// TwinCAT 3 PLC project OSCAT
// Title: AixOCAT
// Company: RWTH Aachen University; E.ON Energy Research Center
// ProjectVersion: 1.0.0
// ProgramVersion: 3.1.4022.1
// project tree:
//   beckhoff_network/Data types/DATA_LOG/ DLOG_DATA.TcDUT, LOG_CONTROL.TcDUT, MYSQL_COM.TcDUT (not stored), PRINTF_DATA.TcDUT (not stored), UNI_CIRCULAR_BUFFER_DATA.TcDUT (not stored), us_LOG_VIEWPORT.TcDUT
//   beckhoff_network/Data types/FILE_SERVER/ FILE_PATH_DATA.TcDUT, FILE_SERVER_DATA.TcDUT
//   beckhoff_network/Data types/NETWORK/ IP2GEO_DATA.TcDUT (not stored), IP_C.TcDUT (not stored), IP_FIFO_DATA.TcDUT (not stored), NETWORK_BUFFER.TcDUT, NETWORK_BUFFER_SHORT.TcDUT (not stored), NW_BUF_LONG.TcDUT (not stored), NW_BUF_SHORT.TcDUT, URL.TcDUT (not stored), VMAP_DATA.TcDUT (not stored), XML_CONTROL.TcDUT (not stored)
//   beckhoff_network/Data types/NET_VAR/ NET_VAR_DATA.TcDUT
//   beckhoff_network/Data types/TELNET_VISION/ us_TN_INPUT_CONTROL.TcDUT, us_TN_INPUT_CONTROL_DATA.TcDUT (not stored), us_TN_MENU.TcDUT, us_TN_MENU_POPUP.TcDUT (not stored), us_TN_SCREEN.TcDUT
//   beckhoff_network/Data types/WEATHER/ WORLD_WEATHER_CUR.TcDUT (not stored), WORLD_WEATHER_DATA.TcDUT, WORLD_WEATHER_DAY.TcDUT (not stored), YAHOO_WEATHER_DATA.TcDUT (not stored)
//   beckhoff_network/Global Variables/ Constants_1.TcGVL, Globale_Variablen_1.TcGVL
//   beckhoff_network/POUs/CO_NVERT/ BASE64_DECODE_STR.TcPOU, BASE64_DECODE_STREAM.TcPOU, BASE64_ENCODE_STR.TcPOU (not stored), BASE64_ENCODE_STREAM.TcPOU, HTML_DECODE.TcPOU (not stored), HTML_ENCODE.TcPOU (not stored), IP4_CHECK.TcPOU, IP4_DECODE.TcPOU (not stored), IP4_TO_STRING.TcPOU, IS_IP4.TcPOU, IS_URLCHR.TcPOU (not stored), MD5_AUX.TcPOU, MD5_CRAM_AUTH.TcPOU (not stored), MD5_STR.TcPOU (not stored), MD5_STREAM.TcPOU (not stored), MD5_TO_STRH.TcPOU, RC4_CRYPT_STREAM.TcPOU (not stored), SHA1_STR.TcPOU, SHA1_STREAM.TcPOU, SHA1_TO_STRH.TcPOU (not stored), STRING_TO_URL.TcPOU (not stored), URL_DECODE.TcPOU (not stored), URL_ENCODE.TcPOU, URL_TO_STRING.TcPOU (not stored)
//   beckhoff_network/POUs/DATA_LOG/ DLOG_BOOL.TcPOU (not stored), DLOG_DINT.TcPOU (not stored), DLOG_DT.TcPOU (not stored), DLOG_FILE_TO_FTP.TcPOU (not stored), DLOG_FILE_TO_SMTP.TcPOU (not stored), DLOG_REAL.TcPOU (not stored), DLOG_STORE_FILE_CSV.TcPOU (not stored), DLOG_STORE_FILE_HTML.TcPOU (not stored), DLOG_STORE_FILE_XML.TcPOU (not stored), DLOG_STORE_RRD.TcPOU (not stored), DLOG_STRING.TcPOU (not stored), UNI_CIRCULAR_BUFFER.TcPOU (not stored)
//   beckhoff_network/POUs/DEMO/ BASE64_DEMO.TcPOU (not stored) (excluded from build), CSV_PARSER_BUF_DEMO.TcPOU (not stored) (excluded from build), CSV_PARSER_FILE_DEMO.TcPOU (excluded from build), DLOG_FILE_CSV_DEMO.TcPOU (not stored) (excluded from build), DLOG_FILE_CSV_FTP_DEMO.TcPOU (not stored) (excluded from build), DLOG_FILE_CSV_SMTP_DEMO.TcPOU (not stored) (excluded from build), DLOG_FILE_HTML_DEMO.TcPOU (not stored) (excluded from build), DLOG_FILE_XML_DEMO.TcPOU (excluded from build), DLOG_RRD_DEMO.TcPOU (not stored) (excluded from build), DNS_DYN_DEMO.TcPOU (excluded from build), DNS_REV_DEMO.TcPOU (not stored) (excluded from build), DNS_SNTP_SYSLOG_DEMO.TcPOU (not stored) (excluded from build), FILE_BLOCK_DEMO.TcPOU (not stored) (excluded from build), FTP_CLIENT_DEMO.TcPOU (excluded from build), GET_WAN_IP_DEMO.TcPOU (excluded from build), HTTP_DEMO.TcPOU (not stored) (excluded from build), INI_PARSER_BUF_DEMO.TcPOU (excluded from build), INI_PARSER_FILE_DEMO.TcPOU (not stored) (excluded from build), IP2GEO_DEMO.TcPOU (excluded from build), IRTRANS_DEMO.TcPOU (not stored) (excluded from build), MB_CLIENT_DEMO.TcPOU (not stored) (excluded from build), MB_SERVER_DEMO.TcPOU (excluded from build), MD5_CRAM_AUTH_DEMO.TcPOU (excluded from build), NET_VAR_MASTER_DEMO.TcPOU (excluded from build), NET_VAR_SLAVE_DEMO.TcPOU (not stored) (excluded from build), RC4_CRYPT_DEMO.TcPOU (not stored) (excluded from build), SHA1_MD5_DEMO.TcPOU (excluded from build), SMTP_CLIENT_DEMO.TcPOU (excluded from build), SPIDER_DEMO.TcPOU (excluded from build), TELNET_LOG_DEMO.TcPOU (excluded from build), TELNET_PRINT_DEMO.TcPOU (not stored) (excluded from build), TN_VISION_DEMO_1.TcPOU (excluded from build), TN_VISION_DEMO_2.TcPOU (not stored) (excluded from build), WORLD_WEATHER_DEMO.TcPOU (not stored) (excluded from build), YAHOO_WEATHER_DEMO.TcPOU (not stored) (excluded from build)
//   beckhoff_network/POUs/DRIVER/ IRTRANS_DECODE.TcPOU (not stored), IRTRANS_RCV_1.TcPOU (not stored), IRTRANS_RCV_4.TcPOU (not stored), IRTRANS_RCV_8.TcPOU (not stored), IRTRANS_SERVER.TcPOU (not stored), IRTRANS_SND_1.TcPOU, IRTRANS_SND_4.TcPOU (not stored), IRTRANS_SND_8.TcPOU (not stored)
//   beckhoff_network/POUs/FILE/ CSV_PARSER_BUF.TcPOU, CSV_PARSER_FILE.TcPOU (not stored), FILE_BLOCK.TcPOU (not stored), FILE_PATH_SPLIT.TcPOU (not stored), INI_PARSER_BUF.TcPOU (not stored), INI_PARSER_FILE.TcPOU (not stored)
//   beckhoff_network/POUs/HARDWARE/ FILE_SERVER.TcPOU, IP_CONTROL.TcPOU, IP_CONTROL2.TcPOU, IP_CONTROL_RESET.TcPOU
//   beckhoff_network/POUs/NETWORK/ DNS_CLIENT.TcPOU, DNS_DYN.TcPOU (not stored), DNS_REV_CLIENT.TcPOU (not stored), FTP_CLIENT.TcPOU, GET_WAN_IP.TcPOU, HTTP_GET.TcPOU (not stored), IP2GEO.TcPOU, IP_FIFO.TcPOU (not stored), LOG_MSG.TcPOU, LOG_VIEWPORT.TcPOU (not stored), MB_CLIENT.TcPOU, MB_SERVER.TcPOU, MB_VMAP.TcPOU, PRINT_SF.TcPOU, READ_HTTP.TcPOU, SMTP_CLIENT.TcPOU, SNTP_CLIENT.TcPOU (not stored), SNTP_SERVER.TcPOU, SPIDER_ACCESS.TcPOU (not stored), SYS_LOG.TcPOU (not stored), TELNET_LOG.TcPOU (not stored), TELNET_PRINT.TcPOU, XML_READER.TcPOU (not stored)
//   beckhoff_network/POUs/NET_VAR/ NET_VAR_BOOL8.TcPOU, NET_VAR_BUFFER.TcPOU, NET_VAR_CONTROL.TcPOU, NET_VAR_DWORD8.TcPOU, NET_VAR_REAL8.TcPOU (not stored), NET_VAR_STRING.TcPOU, NET_VAR_X8.TcPOU
//   beckhoff_network/POUs/OTHER/ ELEMENT_COUNT.TcPOU, ELEMENT_GET.TcPOU (not stored), NETWORK_VERSION.TcPOU (not stored)
//   beckhoff_network/POUs/TELNET_VISION/ TN_FRAMEWORK.TcPOU, TN_INPUT_CONTROL.TcPOU (not stored), TN_INPUT_EDIT_LINE.TcPOU (not stored), TN_INPUT_MENU_BAR.TcPOU, TN_INPUT_MENU_POPUP.TcPOU (not stored), TN_INPUT_SELECT_POPUP.TcPOU (not stored), TN_INPUT_SELECT_TEXT.TcPOU (not stored), TN_RECEIVE.TcPOU (not stored), TN_SC_ADD_SHADOW.TcPOU, TN_SC_AREA_RESTORE.TcPOU, TN_SC_AREA_SAVE.TcPOU (not stored), TN_SC_BOX.TcPOU (not stored), TN_SC_FILL.TcPOU, TN_SC_LINE.TcPOU, TN_SC_READ_ATTR.TcPOU, TN_SC_READ_CHAR.TcPOU, TN_SC_SHADOW_ATTR.TcPOU (not stored), TN_SC_VIEWPORT.TcPOU, TN_SC_WRITE.TcPOU, TN_SC_WRITE_ATTR.TcPOU (not stored), TN_SC_WRITE_C.TcPOU (not stored), TN_SC_WRITE_CHAR.TcPOU (not stored), TN_SC_WRITE_EOS.TcPOU, TN_SC_XY2_ERROR.TcPOU, TN_SC_XY_ERROR.TcPOU (not stored), TN_SEND_ROWS.TcPOU
//   beckhoff_network/POUs/WEATHER/ MOON_PHASE.TcPOU (not stored), WORLD_WEATHER.TcPOU (not stored), WORLD_WEATHER_DESC_GE.TcPOU, WORLD_WEATHER_ICON_OSCAT.TcPOU, YAHOO_WEATHER.TcPOU (not stored), YAHOO_WEATHER_DESC_GE.TcPOU (not stored), YAHOO_WEATHER_ICON_OSCAT.TcPOU
//   oscat_basic/Data types/ CALENDAR.TcDUT, COMPLEX.TcDUT (not stored), CONSTANTS_LANGUAGE.TcDUT (not stored), CONSTANTS_LOCATION.TcDUT (not stored), CONSTANTS_MATH.TcDUT (not stored), CONSTANTS_PHYS.TcDUT (not stored), CONSTANTS_SETUP.TcDUT (not stored), ESR_DATA.TcDUT (not stored), FRACTION.TcDUT (not stored), HOLIDAY_DATA.TcDUT, REAL2.TcDUT (not stored), SDT.TcDUT (not stored), TIMER_EVENT.TcDUT, VECTOR_3.TcDUT (not stored)
//   oscat_basic/Global Variables/ Constants_2.TcGVL (not stored), Globale_Variablen_2.TcGVL, Setup_Data_1.TcGVL
//   oscat_basic/POUs/Buffer Management/ BUFFER_COMP.TcPOU, BUFFER_SEARCH.TcPOU (not stored), BUFFER_TO_STRING.TcPOU (not stored), _BUFFER_CLEAR.TcPOU (not stored), _BUFFER_INIT.TcPOU (not stored), _BUFFER_INSERT.TcPOU (not stored), _BUFFER_UPPERCASE.TcPOU (not stored), _STRING_TO_BUFFER.TcPOU
//   oscat_basic/POUs/Engineering/automation/ DRIVER_1.TcPOU (not stored), DRIVER_4.TcPOU (not stored), DRIVER_4C.TcPOU, FLOW_CONTROL.TcPOU (not stored), FT_Profile.TcPOU, INC_DEC.TcPOU (not stored), INTERLOCK.TcPOU (not stored), INTERLOCK_4.TcPOU (not stored), MANUAL.TcPOU (not stored), MANUAL_1.TcPOU (not stored), MANUAL_2.TcPOU (not stored), MANUAL_4.TcPOU, PARSET.TcPOU, PARSET2.TcPOU (not stored), SIGNAL.TcPOU, SIGNAL_4.TcPOU (not stored), SRAMP.TcPOU, TUNE.TcPOU, TUNE2.TcPOU
//   oscat_basic/POUs/Engineering/Control/ BAND_B.TcPOU, CONTROL_SET1.TcPOU (not stored), CONTROL_SET2.TcPOU (not stored), CTRL_IN.TcPOU (not stored), CTRL_OUT.TcPOU (not stored), CTRL_PI.TcPOU (not stored), CTRL_PID.TcPOU (not stored), CTRL_PWM.TcPOU (not stored), DEAD_BAND.TcPOU, DEAD_BAND_A.TcPOU (not stored), DEAD_ZONE.TcPOU, DEAD_ZONE2.TcPOU (not stored), FB_Integrate.TcPOU (not stored), FB_PID.TcPOU (not stored), FT_DERIV.TcPOU, FT_IMP.TcPOU (not stored), FT_INT.TcPOU, FT_INT2.TcPOU, FT_PD.TcPOU, FT_PDT1.TcPOU, FT_PI.TcPOU (not stored), FT_PID.TcPOU (not stored), FT_PIDW.TcPOU, FT_PIDWL.TcPOU (not stored), FT_PIW.TcPOU (not stored), FT_PIWL.TcPOU, FT_PT1.TcPOU (not stored), FT_PT2.TcPOU, FT_TN16.TcPOU (not stored), FT_TN64.TcPOU (not stored), FT_TN8.TcPOU (not stored), HYST.TcPOU (not stored), HYST_1.TcPOU (not stored), HYST_2.TcPOU (not stored), HYST_3.TcPOU (not stored), INTEGRATE.TcPOU
//   oscat_basic/POUs/Engineering/CO_Nversion/ ASTRO.TcPOU, BFT_TO_MS.TcPOU, C_TO_F.TcPOU (not stored), C_TO_K.TcPOU (not stored), DEG_TO_DIR.TcPOU (not stored), DIR_TO_DEG.TcPOU (not stored), ENERGY.TcPOU (not stored), F_TO_C.TcPOU, F_TO_OM.TcPOU (not stored), F_TO_PT.TcPOU (not stored), GEO_TO_DEG.TcPOU, KMH_TO_MS.TcPOU (not stored), K_TO_C.TcPOU (not stored), LENGTH.TcPOU, MS_TO_BFT.TcPOU (not stored), MS_TO_KMH.TcPOU (not stored), OM_TO_F.TcPOU (not stored), PRESSURE.TcPOU (not stored), PT_TO_F.TcPOU (not stored), SPEED.TcPOU, TEMPERATURE.TcPOU
//   oscat_basic/POUs/Engineering/measurements/ ALARM_2.TcPOU, BAR_GRAPH.TcPOU (not stored), CALIBRATE.TcPOU (not stored), CYCLE_TIME.TcPOU, DT_SIMU.TcPOU, FLOW_METER.TcPOU (not stored), METER.TcPOU (not stored), METER_STAT.TcPOU (not stored), M_D.TcPOU (not stored), M_T.TcPOU, M_TX.TcPOU, ONTIME.TcPOU (not stored), TC_MS.TcPOU (not stored), TC_S.TcPOU, TC_US.TcPOU, T_PLC_MS.TcPOU (not stored), T_PLC_US.TcPOU (not stored)
//   oscat_basic/POUs/Engineering/sensor/ MULTI_IN.TcPOU, RES_NI.TcPOU (not stored), RES_NTC.TcPOU (not stored), RES_PT.TcPOU (not stored), RES_SI.TcPOU, SENSOR_INT.TcPOU, TEMP_NI.TcPOU, TEMP_NTC.TcPOU (not stored), TEMP_PT.TcPOU (not stored), TEMP_SI.TcPOU (not stored)
//   oscat_basic/POUs/Engineering/signal generators/ GEN_PULSE.TcPOU (not stored), GEN_PW2.TcPOU (not stored), GEN_RDM.TcPOU, GEN_RDT.TcPOU, GEN_RMP.TcPOU (not stored), GEN_SIN.TcPOU, GEN_SQR.TcPOU (not stored), PWM_DC.TcPOU (not stored), PWM_PW.TcPOU, RMP_B.TcPOU (not stored), RMP_SOFT.TcPOU (not stored), RMP_W.TcPOU (not stored), _RMP_B.TcPOU (not stored), _RMP_NEXT.TcPOU, _RMP_W.TcPOU
//   oscat_basic/POUs/Engineering/signal processing/ AIN.TcPOU, AIN1.TcPOU (not stored), AOUT.TcPOU (not stored), AOUT1.TcPOU (not stored), BYTE_TO_RANGE.TcPOU (not stored), DELAY.TcPOU (not stored), DELAY_4.TcPOU, FADE.TcPOU (not stored), FILTER_DW.TcPOU (not stored), FILTER_I.TcPOU (not stored), FILTER_MAV_DW.TcPOU, FILTER_MAV_W.TcPOU (not stored), FILTER_W.TcPOU, FILTER_WAV.TcPOU, MIX.TcPOU, MUX_R2.TcPOU, MUX_R4.TcPOU (not stored), OFFSET.TcPOU, OFFSET2.TcPOU (not stored), OVERRIDE.TcPOU (not stored), RANGE_TO_BYTE.TcPOU (not stored), RANGE_TO_WORD.TcPOU (not stored), SCALE.TcPOU, SCALE_B.TcPOU (not stored), SCALE_B2.TcPOU (not stored), SCALE_B4.TcPOU (not stored), SCALE_B8.TcPOU, SCALE_D.TcPOU (not stored), SCALE_R.TcPOU (not stored), SCALE_X2.TcPOU, SCALE_X4.TcPOU (not stored), SCALE_X8.TcPOU, SEL2_OF_3.TcPOU (not stored), SEL2_OF_3B.TcPOU, SH.TcPOU, SH_1.TcPOU (not stored), SH_2.TcPOU (not stored), SH_T.TcPOU (not stored), STAIR.TcPOU, STAIR2.TcPOU, TREND.TcPOU (not stored), TREND_DW.TcPOU, WORD_TO_RANGE.TcPOU (not stored)
//   oscat_basic/POUs/List Processing/ LIST_ADD.TcPOU (not stored), LIST_CLEAN.TcPOU, LIST_GET.TcPOU (not stored), LIST_INSERT.TcPOU (not stored), LIST_LEN.TcPOU (not stored), LIST_NEXT.TcPOU (not stored), LIST_RETRIEVE.TcPOU, LIST_RETRIEVE_LAST.TcPOU
//   oscat_basic/POUs/Logic/FF edge triggered/ COUNT_BR.TcPOU (not stored), COUNT_DR.TcPOU, FF_D2E.TcPOU (not stored), FF_D4E.TcPOU, FF_DRE.TcPOU (not stored), FF_JKE.TcPOU (not stored), FF_RSE.TcPOU, SELECT_8.TcPOU (not stored), SHR_4E.TcPOU, SHR_4UDE.TcPOU (not stored), SHR_8PLE.TcPOU, SHR_8UDE.TcPOU (not stored), TOGGLE.TcPOU (not stored)
//   oscat_basic/POUs/Logic/FF pulse triggered/ LTCH.TcPOU, LTCH_4.TcPOU, STORE_8.TcPOU (not stored)
//   oscat_basic/POUs/Logic/gate logic/ BCDC_TO_INT.TcPOU (not stored), BIT_COUNT.TcPOU (not stored), BIT_LOAD_B.TcPOU (not stored), BIT_LOAD_B2.TcPOU (not stored), BIT_LOAD_DW.TcPOU (not stored), BIT_LOAD_DW2.TcPOU (not stored), BIT_LOAD_W.TcPOU, BIT_LOAD_W2.TcPOU (not stored), BIT_OF_DWORD.TcPOU (not stored), BIT_TOGGLE_B.TcPOU, BIT_TOGGLE_DW.TcPOU (not stored), BIT_TOGGLE_W.TcPOU (not stored), BYTE_OF_BIT.TcPOU, BYTE_OF_DWORD.TcPOU (not stored), BYTE_TO_BITS.TcPOU, BYTE_TO_GRAY.TcPOU (not stored), CHECK_PARITY.TcPOU, CHK_REAL.TcPOU (not stored), DEC_2.TcPOU (not stored), DEC_4.TcPOU (not stored), DEC_8.TcPOU (not stored), DWORD_OF_BYTE.TcPOU (not stored), DWORD_OF_WORD.TcPOU (not stored), DW_TO_REAL.TcPOU (not stored), GRAY_TO_BYTE.TcPOU (not stored), INT_TO_BCDC.TcPOU (not stored), MUX_2.TcPOU (not stored), MUX_4.TcPOU (not stored), PARITY.TcPOU (not stored), REAL_TO_DW.TcPOU (not stored), REFLECT.TcPOU (not stored), REVERSE.TcPOU (not stored), SHL1.TcPOU (not stored), SHR1.TcPOU (not stored), SWAP_BYTE.TcPOU, SWAP_BYTE2.TcPOU (not stored), WORD_OF_BYTE.TcPOU, WORD_OF_DWORD.TcPOU (not stored)
//   oscat_basic/POUs/Logic/generators/ A_TRIG.TcPOU, B_TRIG.TcPOU (not stored), CLICK_CNT.TcPOU (not stored), CLICK_DEC.TcPOU, CLK_DIV.TcPOU, CLK_N.TcPOU (not stored), CLK_PRG.TcPOU (not stored), CLK_PULSE.TcPOU (not stored), CYCLE_4.TcPOU (not stored), D_TRIG.TcPOU (not stored), GEN_BIT.TcPOU, GEN_SQ.TcPOU (not stored), SCHEDULER.TcPOU (not stored), SCHEDULER_2.TcPOU, SEQUENCE_4.TcPOU, SEQUENCE_64.TcPOU (not stored), SEQUENCE_8.TcPOU (not stored), TMAX.TcPOU (not stored), TMIN.TcPOU (not stored), TOF_1.TcPOU (not stored), TONOF.TcPOU (not stored), TP_1.TcPOU (not stored), TP_1D.TcPOU, TP_X.TcPOU (not stored)
//   oscat_basic/POUs/Logic/memory/ FIFO_16.TcPOU, FIFO_32.TcPOU (not stored), STACK_16.TcPOU (not stored), STACK_32.TcPOU (not stored)
//   oscat_basic/POUs/Logic/Others/ CRC_GEN.TcPOU (not stored), MATRIX.TcPOU, PIN_CODE.TcPOU (not stored)
//   oscat_basic/POUs/Mathematical/ ACOSH.TcPOU (not stored), ACOTH.TcPOU, AGDF.TcPOU (not stored), ASINH.TcPOU (not stored), ATAN2.TcPOU (not stored), ATANH.TcPOU, BETA.TcPOU (not stored), BINOM.TcPOU (not stored), CAUCHY.TcPOU (not stored), CAUCHYCD.TcPOU, CEIL.TcPOU, CEIL2.TcPOU, CMP.TcPOU (not stored), COSH.TcPOU (not stored), COTH.TcPOU (not stored), DEC1.TcPOU (not stored), DEG.TcPOU, DIFFER.TcPOU, D_TRUNC.TcPOU (not stored), ERF.TcPOU (not stored), ERFC.TcPOU (not stored), EVEN.TcPOU (not stored), EXP10.TcPOU (not stored), EXPN.TcPOU, FACT.TcPOU, FIB.TcPOU (not stored), FLOOR.TcPOU (not stored), FLOOR2.TcPOU (not stored), FRACT.TcPOU (not stored), GAMMA.TcPOU (not stored), GAUSS.TcPOU (not stored), GAUSSCD.TcPOU (not stored), GCD.TcPOU (not stored), GDF.TcPOU (not stored), GOLD.TcPOU (not stored), HYPOT.TcPOU (not stored), INC.TcPOU (not stored), INC1.TcPOU (not stored), INC2.TcPOU (not stored), INV.TcPOU (not stored), LAMBERT_W.TcPOU (not stored), LANGEVIN.TcPOU (not stored), MAX3.TcPOU (not stored), MID3.TcPOU (not stored), MIN3.TcPOU, MODR.TcPOU (not stored), MUL_ADD.TcPOU (not stored), NEGX.TcPOU (not stored), RAD.TcPOU, RDM.TcPOU, RDM2.TcPOU (not stored), RDMDW.TcPOU (not stored), REAL_TO_FRAC.TcPOU (not stored), RND.TcPOU, ROUND.TcPOU, SGN.TcPOU (not stored), SIGMOID.TcPOU (not stored), SIGN_I.TcPOU (not stored), SIGN_R.TcPOU, SINC.TcPOU (not stored), SINH.TcPOU, SQRTN.TcPOU (not stored), TANC.TcPOU (not stored), TANH.TcPOU (not stored), WINDOW.TcPOU (not stored), WINDOW2.TcPOU (not stored)
//   oscat_basic/POUs/Mathematical/Array/ ARRAY_AVG.TcPOU (not stored), ARRAY_GAV.TcPOU (not stored), ARRAY_HAV.TcPOU (not stored), ARRAY_MAX.TcPOU (not stored), ARRAY_MIN.TcPOU, ARRAY_SDV.TcPOU (not stored), ARRAY_SPR.TcPOU (not stored), ARRAY_SUM.TcPOU (not stored), ARRAY_TREND.TcPOU (not stored), ARRAY_VAR.TcPOU (not stored), IS_SORTED.TcPOU, _ARRAY_ABS.TcPOU, _ARRAY_ADD.TcPOU, _ARRAY_INIT.TcPOU (not stored), _ARRAY_MEDIAN.TcPOU (not stored), _ARRAY_MUL.TcPOU (not stored), _ARRAY_SHUFFLE.TcPOU, _ARRAY_SORT.TcPOU
//   oscat_basic/POUs/Mathematical/Complex/ CABS.TcPOU, CACOS.TcPOU, CACOSH.TcPOU (not stored), CADD.TcPOU (not stored), CARG.TcPOU (not stored), CASIN.TcPOU (not stored), CASINH.TcPOU (not stored), CATAN.TcPOU (not stored), CATANH.TcPOU, CCON.TcPOU (not stored), CCOS.TcPOU (not stored), CCOSH.TcPOU, CDIV.TcPOU (not stored), CEXP.TcPOU (not stored), CINV.TcPOU (not stored), CLOG.TcPOU (not stored), CMUL.TcPOU (not stored), CPOL.TcPOU (not stored), CPOW.TcPOU, CSET.TcPOU (not stored), CSIN.TcPOU, CSINH.TcPOU (not stored), CSQRT.TcPOU (not stored), CSUB.TcPOU (not stored), CTAN.TcPOU (not stored), CTANH.TcPOU (not stored)
//   oscat_basic/POUs/Mathematical/Double Precision/ R2_ABS.TcPOU, R2_ADD.TcPOU (not stored), R2_ADD2.TcPOU (not stored), R2_MUL.TcPOU (not stored), R2_SET.TcPOU (not stored)
//   oscat_basic/POUs/Mathematical/functions/ FRMP_B.TcPOU, FT_AVG.TcPOU, FT_MIN_MAX.TcPOU (not stored), FT_RMP.TcPOU (not stored), F_LIN.TcPOU (not stored), F_LIN2.TcPOU, F_POLY.TcPOU (not stored), F_POWER.TcPOU (not stored), F_QUAD.TcPOU, LINEAR_INT.TcPOU, POLYNOM_INT.TcPOU (not stored)
//   oscat_basic/POUs/Mathematical/Geometry/ CIRCLE_A.TcPOU (not stored), CIRCLE_C.TcPOU (not stored), CIRCLE_SEG.TcPOU (not stored), CONE_V.TcPOU (not stored), ELLIPSE_A.TcPOU, ELLIPSE_C.TcPOU (not stored), SPHERE_V.TcPOU, TRIANGLE_A.TcPOU (not stored)
//   oscat_basic/POUs/Mathematical/Vektormathematik/ V3_ABS.TcPOU (not stored), V3_ADD.TcPOU (not stored), V3_ANG.TcPOU, V3_DPRO.TcPOU (not stored), V3_NORM.TcPOU, V3_NUL.TcPOU (not stored), V3_PAR.TcPOU (not stored), V3_REV.TcPOU (not stored), V3_SMUL.TcPOU (not stored), V3_SUB.TcPOU (not stored), V3_XANG.TcPOU (not stored), V3_XPRO.TcPOU (not stored), V3_YANG.TcPOU (not stored), V3_ZANG.TcPOU
//   oscat_basic/POUs/Other/ ESR_COLLECT.TcPOU (not stored), ESR_MON_B8.TcPOU, ESR_MON_R4.TcPOU (not stored), ESR_MON_X8.TcPOU, OSCAT_VERSION.TcPOU, STATUS_TO_ESR.TcPOU (not stored)
//   oscat_basic/POUs/String/ BIN_TO_BYTE.TcPOU, BIN_TO_DWORD.TcPOU (not stored), BYTE_TO_STRB.TcPOU (not stored), BYTE_TO_STRH.TcPOU (not stored), CAPITALIZE.TcPOU (not stored), CHARCODE.TcPOU (not stored), CHARNAME.TcPOU (not stored), CHR_TO_STRING.TcPOU, CLEAN.TcPOU, CODE.TcPOU, COUNT_CHAR.TcPOU (not stored), COUNT_SUBSTRING.TcPOU (not stored), DEC_TO_BYTE.TcPOU, DEC_TO_DWORD.TcPOU (not stored), DEC_TO_INT.TcPOU, DEL_CHARS.TcPOU (not stored), DT_TO_STRF.TcPOU, DWORD_TO_STRB.TcPOU (not stored), DWORD_TO_STRF.TcPOU, DWORD_TO_STRH.TcPOU, EXEC.TcPOU (not stored), FILL.TcPOU (not stored), FINDB.TcPOU, FINDB_NONUM.TcPOU (not stored), FINDB_NUM.TcPOU, FINDP.TcPOU (not stored), FIND_CHAR.TcPOU (not stored), FIND_CTRL.TcPOU (not stored), FIND_NONUM.TcPOU, FIND_NUM.TcPOU (not stored), FIX.TcPOU (not stored), FLOAT_TO_REAL.TcPOU (not stored), FSTRING_TO_BYTE.TcPOU (not stored), FSTRING_TO_DT.TcPOU (not stored), FSTRING_TO_DWORD.TcPOU (not stored), FSTRING_TO_MONTH.TcPOU (not stored), FSTRING_TO_WEEK.TcPOU (not stored), FSTRING_TO_WEEKDAY.TcPOU, HEX_TO_BYTE.TcPOU (not stored), HEX_TO_DWORD.TcPOU (not stored), ISC_ALPHA.TcPOU (not stored), ISC_CTRL.TcPOU, ISC_HEX.TcPOU (not stored), ISC_LOWER.TcPOU, ISC_NUM.TcPOU (not stored), ISC_UPPER.TcPOU (not stored), IS_ALNUM.TcPOU (not stored), IS_ALPHA.TcPOU, IS_CC.TcPOU (not stored), IS_CTRL.TcPOU (not stored), IS_HEX.TcPOU (not stored), IS_LOWER.TcPOU (not stored), IS_NCC.TcPOU, IS_NUM.TcPOU (not stored), IS_UPPER.TcPOU (not stored), LOWERCASE.TcPOU, MESSAGE_4R.TcPOU (not stored), MESSAGE_8.TcPOU (not stored), MIRROR.TcPOU (not stored), MONTH_TO_STRING.TcPOU (not stored), OCT_TO_BYTE.TcPOU (not stored), OCT_TO_DWORD.TcPOU, REAL_TO_STRF.TcPOU (not stored), REPLACE_ALL.TcPOU, REPLACE_CHARS.TcPOU (not stored), REPLACE_UML.TcPOU (not stored), TICKER.TcPOU (not stored), TO_LOWER.TcPOU (not stored), TO_UML.TcPOU (not stored), TO_UPPER.TcPOU, TRIM.TcPOU (not stored), TRIM1.TcPOU, TRIME.TcPOU (not stored), UPPERCASE.TcPOU (not stored), WEEKDAY_TO_STRING.TcPOU (not stored)
//   oscat_basic/POUs/Time&Date/ CALENDAR_CALC.TcPOU (not stored), DATE_ADD.TcPOU (not stored), DAYS_DELTA.TcPOU (not stored), DAYS_IN_MONTH.TcPOU (not stored), DAYS_IN_YEAR.TcPOU, DAY_OF_DATE.TcPOU, DAY_OF_MONTH.TcPOU (not stored), DAY_OF_WEEK.TcPOU, DAY_OF_YEAR.TcPOU (not stored), DAY_TO_TIME.TcPOU (not stored), DCF77.TcPOU, DST.TcPOU (not stored), DT2_TO_SDT.TcPOU (not stored), DT_TO_SDT.TcPOU (not stored), EASTER.TcPOU, EVENTS.TcPOU, HOLIDAY.TcPOU (not stored), HOUR.TcPOU (not stored), HOUR_OF_DT.TcPOU, HOUR_TO_TIME.TcPOU (not stored), HOUR_TO_TOD.TcPOU (not stored), JD2000.TcPOU, LEAP_DAY.TcPOU (not stored), LEAP_OF_DATE.TcPOU, LEAP_YEAR.TcPOU (not stored), LTIME_TO_UTC.TcPOU (not stored), MINUTE.TcPOU, MINUTE_OF_DT.TcPOU (not stored), MINUTE_TO_TIME.TcPOU (not stored), MONTH_BEGIN.TcPOU (not stored), MONTH_END.TcPOU, MONTH_OF_DATE.TcPOU (not stored), MULTIME.TcPOU (not stored), PERIOD.TcPOU (not stored), PERIOD2.TcPOU (not stored), REFRACTION.TcPOU (not stored), RTC_2.TcPOU (not stored), RTC_MS.TcPOU (not stored), SDT_TO_DATE.TcPOU (not stored), SDT_TO_DT.TcPOU, SDT_TO_TOD.TcPOU (not stored), SECOND.TcPOU (not stored), SECOND_OF_DT.TcPOU (not stored), SECOND_TO_TIME.TcPOU (not stored), SET_DATE.TcPOU, SET_DT.TcPOU (not stored), SET_TOD.TcPOU (not stored), SUN_MIDDAY.TcPOU (not stored), SUN_POS.TcPOU (not stored), SUN_TIME.TcPOU (not stored), TIMECHECK.TcPOU (not stored), UTC_TO_LTIME.TcPOU, WORK_WEEK.TcPOU (not stored), YEAR_BEGIN.TcPOU, YEAR_END.TcPOU (not stored), YEAR_OF_DATE.TcPOU (not stored)
//   oscat_building/Global Variables/ Constants.TcGVL (not stored), Globale_Variablen.TcGVL, Setup_Data.TcGVL (not stored)
//   oscat_building/POUs/actuators/ ACTUATOR_2P.TcPOU, ACTUATOR_3P.TcPOU, ACTUATOR_A.TcPOU, ACTUATOR_COIL.TcPOU (not stored), ACTUATOR_PUMP.TcPOU, ACTUATOR_UD.TcPOU (not stored), AUTORUN.TcPOU (not stored)
//   oscat_building/POUs/electrical/ CLICK.TcPOU (not stored), CLICK_MODE.TcPOU (not stored), DEBOUNCE.TcPOU, DIMM_2.TcPOU, DIMM_I.TcPOU (not stored), F_LAMP.TcPOU (not stored), PULSE_LENGTH.TcPOU (not stored), PULSE_T.TcPOU, SWITCH_I.TcPOU (not stored), SWITCH_X.TcPOU, SW_RECONFIG.TcPOU (not stored), TIMER_1.TcPOU (not stored), TIMER_2.TcPOU (not stored), TIMER_EVENT_DECODE.TcPOU, TIMER_EXT.TcPOU (not stored), TIMER_P4.TcPOU (not stored)
//   oscat_building/POUs/HLK/ AIR_DENSITY.TcPOU, AIR_ENTHALPY.TcPOU (not stored), BOILER.TcPOU (not stored), BURNER.TcPOU, DEW_CON.TcPOU (not stored), DEW_RH.TcPOU (not stored), DEW_TEMP.TcPOU, HEAT_INDEX.TcPOU (not stored), HEAT_METER.TcPOU (not stored), HEAT_TEMP.TcPOU (not stored), LEGIONELLA.TcPOU, SDD.TcPOU, SDD_NH3.TcPOU, SDT_NH3.TcPOU, TANK_LEVEL.TcPOU, TANK_VOL1.TcPOU, TANK_VOL2.TcPOU (not stored), TEMP_EXT.TcPOU, T_AVG24.TcPOU (not stored), WATER_CP.TcPOU, WATER_DENSITY.TcPOU, WATER_ENTHALPY.TcPOU (not stored), WCT.TcPOU (not stored)
//   oscat_building/POUs/Jalousie/ BLIND_ACTUATOR.TcPOU, BLIND_CONTROL.TcPOU (not stored), BLIND_CONTROL_S.TcPOU (not stored), BLIND_INPUT.TcPOU (not stored), BLIND_NIGHT.TcPOU (not stored), BLIND_SCENE.TcPOU (not stored), BLIND_SECURITY.TcPOU (not stored), BLIND_SET.TcPOU, BLIND_SHADE.TcPOU, BLIND_SHADE_S.TcPOU
//   oscat_building/POUs/Other/ BUILDING_VERSION.TcPOU (not stored)

// ---- beckhoff_network/Data types/DATA_LOG/DLOG_DATA.TcDUT
TYPE DLOG_DATA :
STRUCT
	STORE_TYPE : BYTE;
	ADD_HEADER : BOOL;
	ADD_DATA : BOOL;
	ADD_DATA_REQ : BOOL;
	CLOCK_TRIG : BOOL;
	ID_MAX : USINT;
	DTI : DT;
	UCB : UNI_CIRCULAR_BUFFER_DATA;
	NEW_FILE : STRING;
	NEW_FILE_RTRIG : BOOL;
END_STRUCT
END_TYPE

// ---- beckhoff_network/Data types/DATA_LOG/LOG_CONTROL.TcDUT
TYPE LOG_CONTROL :
STRUCT
	NEW_MSG : STRING(LOG_SIZE); (* neue Nachricht für den Datenbuffer *)
	NEW_MSG_OPTION : DWORD;
	LEVEL : BYTE;
	SIZE : INT := LOG_MAX; (* Anzahl der Strings im LOG_DATA *)
	RESET : BOOL; (* Nachrichtenbuffer löschen *)
	PRINTF : PRINTF_DATA; (* Array PRINTF Parameter *)
	MSG : ARRAY [0..LOG_MAX] OF STRING(LOG_SIZE); (* Array Message *)
	MSG_OPTION : ARRAY [0..LOG_MAX] OF DWORD; (* Array Options *)
	UPDATE_COUNT : UINT; (* Updatezähler *)
	IDX : INT; (* aktueller Nachrichten-Index *)
	RING_MODE : BOOL; (* Bufferüberlauf erkannt *)
END_STRUCT
END_TYPE

// ---- beckhoff_network/Data types/DATA_LOG/us_LOG_VIEWPORT.TcDUT
TYPE us_LOG_VIEWPORT :
STRUCT
	LINE_ARRAY : ARRAY [1..40] OF INT;
	COUNT : INT; (* Anzahl der sichtbaren Nachtrichten *)
	UPDATE_COUNT : UINT; (* Updatezähler *)
	MOVE_TO_X : INT; (* Steuerung der Nachrichtenanzeige *)
	UPDATE : BOOL; (* Daten wurden geändert -> neuzeichnen *)
END_STRUCT
END_TYPE

// ---- beckhoff_network/Data types/FILE_SERVER/FILE_PATH_DATA.TcDUT
TYPE FILE_PATH_DATA :
STRUCT
	DRIVE : STRING(3);
	DIRECTORY : STRING(STRING_LENGTH);
	FILENAME : STRING;
END_STRUCT
END_TYPE

// ---- beckhoff_network/Data types/FILE_SERVER/FILE_SERVER_DATA.TcDUT
TYPE FILE_SERVER_DATA :
STRUCT
	FILE_OPEN : BOOL;
	FILENAME : STRING;
	MODE : BYTE;
	OFFSET : UDINT;
	FILE_SIZE : UDINT;
	AUTO_CLOSE : TIME;
	ERROR : BYTE;
END_STRUCT
END_TYPE

// ---- beckhoff_network/Data types/NETWORK/NETWORK_BUFFER.TcDUT
TYPE NETWORK_BUFFER :
STRUCT
	SIZE : UINT;
	BUFFER : NW_BUF_LONG;
END_STRUCT
END_TYPE

// ---- beckhoff_network/Data types/NETWORK/NW_BUF_SHORT.TcDUT
TYPE
	NW_BUF_SHORT : ARRAY[0..NETWORK_BUFFER_SHORT_SIZE] OF BYTE;
END_TYPE

// ---- beckhoff_network/Data types/NET_VAR/NET_VAR_DATA.TcDUT
TYPE NET_VAR_DATA :
STRUCT
	CYCLE : UDINT;
	STATE : BYTE;
	INDEX : INT;
	ID_MAX : USINT;
	ERROR_ID : BYTE;
	BUF_SIZE : UINT;
	S_BUF : NETWORK_BUFFER;
	R_BUF : NETWORK_BUFFER;
END_STRUCT
END_TYPE

// ---- beckhoff_network/Data types/TELNET_VISION/us_TN_INPUT_CONTROL.TcDUT
TYPE us_TN_INPUT_CONTROL :
STRUCT
	bo_Enable: BOOL; (* Bearbeitung freigeben/sperren *)
	bo_Update_all: BOOL; (* All Elemente neu zeichnen *)
	bo_Reset_Fokus: BOOL; (* Fokus auf 1. Element setzen *)
	in_Focus_at: INT; (* Controlelement mit aktivem Fokus *)
	in_Count: INT; (* Anzahl der benutzen Control-Elemente *)
	in_ToolTip_X: INT; (* Tooltip Text X-Offset *)
	in_ToolTip_Y: INT; (* Tooltip Text Y-Offset *)
	by_ToolTip_Attr: BYTE; (* Tooltip Text Attribute *)
	in_ToolTip_Size: INT; (* Tooltip Text länge *)
	usa_TN_INPUT_CONTROL_DATA: ARRAY [1..20] OF us_TN_INPUT_CONTROL_DATA;
END_STRUCT
END_TYPE

// ---- beckhoff_network/Data types/TELNET_VISION/us_TN_MENU.TcDUT
TYPE us_TN_MENU :
STRUCT
	st_Menu_Text: STRING(STRING_LENGTH); (* X Menue Texte *)
	in_Menu_E_Count: INT; (* Menue Elemente Anzahl *)
	in_Y: INT; (* Menue Zeilennummer  Y-Position *)
	in_X: INT; (* Menue Spaltennummer X-Position *)
	by_Attr_mF: BYTE; (* Text Attribute mit Fokus *)
	by_Attr_oF: BYTE; (* Text Attribute ohne Fokus *)
	in_X_SM_new: INT; (* neue Sub-Menu X-Position *)
	in_Y_SM_new: INT; (* neue Sub-Menu Y-Position *)
	in_X_SM_old: INT; (* alte Sub-Menu X-Position *)
	in_Y_SM_old: INT; (* alte Sub-Menu Y-Position *)
	in_Cur_Menu_Item: INT; (* aktuelles Haupt-Menue *)
	in_Cur_Sub_Item: INT; (* aktuelles Sub-Menue *)
	in_State: INT; (*   Menu status   *)
	in_Menu_Selected: INT; (* X Menu-Item mit Enter angewwählt *)
	bo_Create: BOOL; (* X Menu erzeugen *)
	bo_Destroy: BOOL; (* X Menu entfernen *)
	bo_Update: BOOL; (* X Menu updaten *)
END_STRUCT
END_TYPE

// ---- beckhoff_network/Data types/TELNET_VISION/us_TN_SCREEN.TcDUT
TYPE us_TN_SCREEN :
STRUCT
	bya_CHAR: ARRAY [0..1919] OF BYTE;
	bya_COLOR: ARRAY [0..1919] OF BYTE;
	bya_BACKUP: ARRAY [0..1919] OF BYTE;
	bya_Line_Update: ARRAY [0..23] OF BOOL;
	by_Input_Exten_Code: BYTE;
	by_Input_ASCII_Code: BYTE;
	bo_Input_ASCII_IsNum: BOOL;
	in_Page_Number: INT; (* aktive Seiten-Nr. *)
	in_Cursor_X: INT; (* Cursor X-Position *)
	in_Cursor_Y: INT; (* Cursor Y-Position *)
	in_EOS_Offset: INT; (* End of String Offset *)
	by_Clear_Screen_Attr: BYTE; (* Clear-Screen Attr *)
	bo_Clear_Screen: BOOL; (* Clear-Screen auslösen *)
	bo_Modal_Dialog: BOOL; (* Modaler Dialog ist aktiv *)
	bo_Menue_Bar_Dialog: BOOL; (* Menue Dialog ist aktiv *)
END_STRUCT
END_TYPE

// ---- beckhoff_network/Data types/WEATHER/WORLD_WEATHER_DATA.TcDUT
TYPE WORLD_WEATHER_DATA :
STRUCT
	CUR : WORLD_WEATHER_CUR;
	DAY : ARRAY [0..4] OF WORLD_WEATHER_DAY;
END_STRUCT
END_TYPE

// ---- oscat_basic/Data types/CALENDAR.TcDUT
TYPE CALENDAR :
STRUCT
	UTC : DT;					(* world time UTC *)
	LDT : DT;					(* local time *)
	LDATE : DATE;				(* local date *)
	LTOD : TOD;					(* local time of day *)
	YEAR : INT;					(* year of LDATE *)
	MONTH : INT;				(* month of LDATE *)
	DAY : INT;					(* day of LDATE *)
	WEEKDAY : INT;				(* weekday of LDATE *)
	OFFSET : INT;				(* Time Zone Offset for Local time in minutes *)
	DST_EN : BOOL;				(* daylight savings time enable *)
	DST_ON : BOOL;				(* true when daylight savings time os on *)
	NAME : STRING(5);			(* name of time zone *)
	LANGUAGE : INT;			(* location number pls see location setup *)
	LONGITUDE : REAL;			(* longitude of current location *)
	LATITUDE : REAL;			(* latitude of current location *)
	SUN_RISE : TOD;				(* sun_rise for current location *)
	SUN_SET : TOD;				(* sun_set for current location *)
	SUN_MIDDAY : TOD;			(* worldtime when sun stands at south position *)
	SUN_HEIGTH : REAL	;		(* suns heigth at midday, south position *)
	SUN_HOR : REAL;			(* sun angle horizontal 0 = north in degrees *)
	SUN_VER : REAL;			(* sun angle vertical above horizon in degrees *)
	NIGHT : BOOL;				(* true between sun_set and sun_rise *)
	HOLIDAY : BOOL;			(* true when holiday *)
	HOLY_NAME : STRING(30);	(* name of holiday *)
	WORK_WEEK : INT;			(* current work week *)
END_STRUCT
END_TYPE

// ---- oscat_basic/Data types/HOLIDAY_DATA.TcDUT
TYPE HOLIDAY_DATA :
STRUCT
	NAME : STRING(30);
	DAY : SINT;
	MONTH : SINT;
	USE : SINT;
END_STRUCT
END_TYPE

// ---- oscat_basic/Data types/TIMER_EVENT.TcDUT
TYPE TIMER_EVENT :
STRUCT
	TYP : BYTE;
	CHANNEL : BYTE;
	DAY : BYTE;
	START : TOD;
	DURATION : TIME;
	LAND : BYTE;
	LOR : BYTE;
	LAST : DT;
END_STRUCT
END_TYPE

// ---- beckhoff_network/Global Variables/Constants_1.TcGVL
{attribute 'Tc2GvlVarNames'}
VAR_GLOBAL CONSTANT
	NETWORK_BUFFER_LONG_SIZE : UINT := 4095;
	NETWORK_BUFFER_SHORT_SIZE : UINT := 1407;
	LOG_MAX : INT := 40;
	LOG_SIZE : INT := 80;
	ELEMENT_LENGTH : INT := 250;
END_VAR

// ---- beckhoff_network/Global Variables/Globale_Variablen_1.TcGVL
{attribute 'Tc2GvlVarNames'}
VAR_GLOBAL
	TCP_SERVER_RESET : BYTE; (* nur für TwinCAT notwendig ! *)
	LOG_CL : LOG_CONTROL;
END_VAR

// ---- oscat_basic/Global Variables/Globale_Variablen_2.TcGVL
{attribute 'Tc2GvlVarNames'}
VAR_GLOBAL
	MATH : CONSTANTS_MATH;
	PHYS : CONSTANTS_PHYS;
	LANGUAGE : CONSTANTS_LANGUAGE;
	SETUP : CONSTANTS_SETUP;
	LOCATION : CONSTANTS_LOCATION;
END_VAR

// ---- oscat_basic/Global Variables/Setup_Data_1.TcGVL
{attribute 'Tc2GvlVarNames'}
VAR_GLOBAL RETAIN

END_VAR

// ---- oscat_building/Global Variables/Globale_Variablen.TcGVL
{attribute 'Tc2GvlVarNames'}
VAR_GLOBAL
END_VAR

// ---- beckhoff_network/POUs/CO_NVERT/BASE64_DECODE_STR.TcPOU
FUNCTION_BLOCK BASE64_DECODE_STR
VAR_INPUT
	RUN : BOOL;
END_VAR
VAR_OUTPUT
	DONE : BOOL;
END_VAR
VAR_IN_OUT
	STR1 : STRING(192);
	STR2 : STRING(144);
END_VAR
VAR
	BASE64_DECODE_STREAM : BASE64_DECODE_STREAM;
	run_last : BOOL;
	buf1 : ARRAY [0..63] OF BYTE;
	buf2 : ARRAY [0..47] OF BYTE;
	mode : INT;
	size1 : INT;
	size2 : INT;
	end : INT;
	pos : INT;
END_VAR

(*
version 1.0	06. dec. 2009
programmer 	ks
tested by	ks

BASE64_DECODE_STR konvertiert einen BASE64 kodierten String in einen normalen String. 

*)

CASE mode OF
0:	IF RUN AND NOT run_last THEN
		DONE := FALSE;
		mode := 1;
		end := LEN(STR1);
		pos := 0;
		STR2 := '';
	END_IF;
1:
	size1 := MIN(48,end - pos);
	IF size1 > 0 THEN
		_STRING_TO_BUFFER(STR:=MID(STR1, size1, pos + 1), POS:=0, PT:=ADR(buf1), SIZE:=SIZEOF(buf1));
		BASE64_DECODE_STREAM(BUF1:=buf1 ,BUF2:=buf2 ,SIZE1:=size1 ,SIZE2=>size2);
		STR2 := CONCAT(STR2,BUFFER_TO_STRING(PT:=ADR(buf2), SIZE:=SIZEOF(buf2), START:=0, STOP:=size2 - 1));
	ELSE
		mode := 0;
		DONE := TRUE;
	END_IF;
	pos := pos + size1;
END_CASE;

run_last := RUN;

(* revision history

ks	6. dec. 2009 rev 1.0
	original version

*)

END_FUNCTION_BLOCK

// ---- beckhoff_network/POUs/CO_NVERT/BASE64_DECODE_STREAM.TcPOU
FUNCTION_BLOCK BASE64_DECODE_STREAM
VAR_IN_OUT
	BUF1 : ARRAY [0..63] OF BYTE;
	BUF2 : ARRAY [0..47] OF BYTE;
END_VAR
VAR_INPUT
	SIZE1 : INT;
END_VAR
VAR_OUTPUT
	SIZE2 : INT;
END_VAR
VAR_TEMP
	a: INT;
	b: WORD;
	o: INT;
	off: INT;
	i1: INT;
	i2: INT;
	c: INT;
END_VAR

(*
version 1.0	06. dec. 2009
programmer 	ks
tested by	ks

BASE64_DECODE_STREAM konvertiert einzelne Base64 kodierte Datenblöcke in normalen Datenblöcke. 

*)

IF SIZE1 <= 0 THEN SIZE2 := 0; RETURN; END_IF;
c := SIZE1 - 1;
i2 := 0;
a := 0;
b := 0;
FOR i1 := 0 TO c DO
	o := BUF1[i1];
	IF o = 61  (* = *) THEN	EXIT;
	ELSIF o > 96 (* a-z *) THEN off := 71;
	ELSIF o > 64 (* A-Z *) THEN off := 65;
	ELSIF o > 47 (* 0-9 *) THEN off := -4;
	ELSIF o = 43 (* + *) THEN off := -19;
	ELSIF o = 47 (* / *) THEN off := -16;
	END_IF;
	b := SHL(b,6) OR INT_TO_BYTE(o - off);
	a := a + 6;
	IF a >= 8 THEN
		a := a - 8;
		BUF2[i2] := WORD_TO_BYTE(SHR(b,a));
		i2 := i2 + 1;
		b := b AND NOT SHL(WORD#16#FFFF,a);
	END_IF;
END_FOR;
SIZE2 := i2;

(* revision history

ks	6. dec. 2009 rev 1.0
	original version

*)

END_FUNCTION_BLOCK

// ---- oscat_basic/POUs/Buffer Management/_STRING_TO_BUFFER.TcPOU
FUNCTION _STRING_TO_BUFFER : INT
VAR_INPUT
	STR : STRING(STRING_LENGTH);
	POS : INT;
	PT : POINTER TO ARRAY[0..32767] OF BYTE;
	SIZE : UINT;
END_VAR
VAR
	ps : POINTER TO BYTE;
	i: INT;
	end: INT;
END_VAR


(*
version 1.4	2. jan. 2012
programmer 	hugo
tested by		oscat

this function will copy a string into an array of byte starting at position pos.
the function needs to be called:	_String_To_buffer(str, pos, adr("array"),sizeof("array"));
this function will manipulate the array directly in memory and returns the position after the input string when finished.
because this function works with pointers its very time efficient and it needs no extra memory.

*)

ps := ADR(str);
end := MIN(pos + LEN(str), UINT_TO_INT(size));
IF end > 0 THEN end := end -1; END_IF;
FOR i := pos TO end DO
	pt^[i] := ps^;
	ps := ps + 1;
END_FOR;

_STRING_TO_BUFFER := i;

(* revision History

hm 	5. mar. 2008	rev 1.0
	original version

hm	16. mar. 2008	rev 1.1
	changed type of input size to uint

hm	13. may. 2008	rev 1.2
	changed type of pointer to array[1..32767]
	changed size of string to STRING_LENGTH

hm	12. nov. 2009	rev 1.3
	limit end to size - 1

hm	2. jan 2012	rev 1.4
	return the position after the input string when finished
*)

END_FUNCTION

// ---- beckhoff_network/POUs/CO_NVERT/BASE64_ENCODE_STREAM.TcPOU
FUNCTION_BLOCK BASE64_ENCODE_STREAM
VAR_IN_OUT
	BUF1 : ARRAY [0..47] OF BYTE;
	BUF2 : ARRAY [0..63] OF BYTE;
END_VAR
VAR_INPUT
	SIZE1 : INT;
END_VAR
VAR_OUTPUT
	SIZE2 : INT;
END_VAR
VAR
	a: INT;
	b: WORD;
	i: INT;
	i2: INT;
	i3: INT;
	c: INT;
	BASE64: STRING(64) := 'ABCDEFGHIJKLMNOPQRSTUVWXYZabcdefghijklmnopqrstuvwxyz0123456789+/';
END_VAR

(*
version 1.0	06. dec. 2009
programmer 	ks
tested by	ks

BASE64_ENCODE_STREAM konvertiert Datenblöcke in Base64. 

*)

IF SIZE1 <= 0 THEN
	SIZE2 := 0;
	RETURN;
END_IF;
c := SIZE1 - 1;
i2 := 0;
a := 0;
b := 0;
FOR i := 0 TO c DO
	b := SHL(b,8) OR BUF1[i];
	a := a + 8;
	WHILE a >= 6 DO
		a := a - 6;
		buf2[i2] := CODE(BASE64,WORD_TO_INT(SHR(b,a)) + 1);
		i2 := i2 + 1;
		b := b AND NOT SHL(WORD#16#FFFF,a);
	END_WHILE;
END_FOR;
IF a > 0 THEN
	buf2[i2] := CODE(BASE64,WORD_TO_INT(SHL(b,6 - a)) + 1);
	i2 := i2 + 1;
	i3 := i2 + (NOT INT_TO_WORD(i2) AND 2#11);
	FOR i := i2 TO i3 DO
		buf2[i] := 61;
	END_FOR;
	SIZE2 := i3 + 1;
ELSE
	SIZE2 := i2;
END_IF;

(* revision history

ks	6. dec. 2009 rev 1.0
	original version

*)

END_FUNCTION_BLOCK

// ---- oscat_basic/POUs/String/CODE.TcPOU
FUNCTION CODE : BYTE
VAR_INPUT
	STR : STRING(STRING_LENGTH);
	POS : INT;
END_VAR
VAR
	PT : POINTER TO BYTE;
END_VAR

(*
version 1.1	29. mar. 2008
programmer 	hugo
tested by		tobias

code extracts the code of a character at position POS of a string STR.

*)

IF pos < 1 OR pos > LEN(str) THEN
	CODE := 0;
	RETURN;
ELSE
	PT := ADR(STR) + INT_TO_DWORD(pos - 1);
	CODE := pt^;
END_IF;

(* revision history
hm	9. mar. 2008	rev 1.0
	original version

hm	29. mar. 2008	rev 1.1
	changed STRING to STRING(STRING_LENGTH)
*)

END_FUNCTION

// ---- beckhoff_network/POUs/CO_NVERT/IP4_CHECK.TcPOU
FUNCTION IP4_CHECK : BOOL
VAR_INPUT
	NIP : DWORD;
	LIP : DWORD;
	SM : DWORD;
END_VAR


(*
version 1.0	4. mar 2008
programmer 	hugo
tested by		oscat

IP4_CHECK testet ob eine Network IP und Local_IP im selben Subnet sind.

*)

IP4_CHECK := (NIP AND sm) = (LIP AND SM);


(* revision history
hm		4. mar 2008	rev 1.0
	original version

*)

END_FUNCTION

// ---- beckhoff_network/POUs/CO_NVERT/IP4_TO_STRING.TcPOU
FUNCTION IP4_TO_STRING : STRING(15)
VAR_INPUT
	IP4 : DWORD;
END_VAR
VAR
	tmp : STRING(3);
END_VAR

(*
version 1.1	10. mar. 2009
programmer 	kurt
tested by	hugo

IP4_TO_STRING erzeugt eine IP Adresse als String aus einem DWORD..

*)

(* mask bits AND INSERT AT given position *)
tmp := BYTE_TO_STRING(DWORD_TO_BYTE(IP4));
IP4_TO_STRING := CONCAT('...', tmp);
tmp := BYTE_TO_STRING(DWORD_TO_BYTE(SHR(IP4,8)));
IP4_TO_STRING := INSERT(IP4_TO_STRING, tmp, 2);
tmp := BYTE_TO_STRING(DWORD_TO_BYTE(SHR(IP4,16)));
IP4_TO_STRING := INSERT(IP4_TO_STRING, tmp, 1);
tmp := BYTE_TO_STRING(DWORD_TO_BYTE(SHR(IP4,24)));
IP4_TO_STRING := CONCAT(tmp, IP4_TO_STRING);



(* revision history
hm	22. apr 2008	rev 1.0
	original version

hm	10. mar. 2009	rev 1.1
	improved code
*)

END_FUNCTION

// ---- beckhoff_network/POUs/CO_NVERT/IS_IP4.TcPOU
FUNCTION IS_IP4 : BOOL
VAR_INPUT
	str : STRING;
END_VAR


(*
version 1.1	10. mar 2009
programmer 	kurt
tested by		hugo

IS_IP4 testet ob ein string eine gültige IPv4 Adresse enthält.

*)

IS_IP4 := COUNT_CHAR(str, 46) = 3;


(* revision history
hm	1. mar. 2008	rev 1.0
	original version

hm	10. mar. 2009	rev 1.1
	new code

*)

END_FUNCTION

// ---- beckhoff_network/POUs/CO_NVERT/MD5_AUX.TcPOU
FUNCTION MD5_AUX : DWORD
VAR_INPUT
	N : INT;
	A : DWORD;
	B : DWORD;
	C : DWORD;
	D : DWORD;
	X : DWORD;
	U : INT;
	T : DWORD;
END_VAR
VAR
	w : DWORD;
END_VAR

(*
version 1.0	06. dec. 2009
programmer 	ks
tested by	ks

MD5_AUX ist ein Zusatzbaustein füR MD5_STREAM und enthäLT wiederkehrende Berechnungen
*)

CASE N OF
	1: w := (B AND C) OR (NOT(B) AND D);
	2: w := (B AND D) OR (C AND NOT D);
	3: w := (B XOR C XOR D);
	4: w := (C XOR (B OR  NOT(D)));
END_CASE

MD5_AUX := B + ROL(A + w + X + T,U);

(* revision history

ks	6. dec. 2009 rev 1.0
	original version

*)

END_FUNCTION

// ---- beckhoff_network/POUs/CO_NVERT/MD5_TO_STRH.TcPOU
FUNCTION MD5_TO_STRH : STRING(32)
VAR_INPUT
	MD5 : ARRAY [0..15] OF BYTE;
END_VAR
VAR
	i : INT;
	tmp : BYTE;
	pt : POINTER TO BYTE;
END_VAR
(*
version 1.0	06. dec. 2009
programmer 	ks
tested BY	ks

MD5_TO_STRH konvertiert das MD5 Hash Array in einen HEX-String
*)

pt := ADR(MD5_TO_STRH); (* read output adress to pointer *)

FOR i := 0 TO 15 DO; (* write the 8 hex characters backwards *)
	tmp := SHR(MD5[i],4);
	PT^ := tmp + SEL(tmp <= 9,87,48);
	pt := pt + 1; (* decrement the pointer *)
	tmp := MD5[i] AND 2#1111;
	PT^ := tmp + SEL(tmp <= 9,87,48);
	pt := pt + 1; (* decrement the pointer *)
END_FOR;
pt^:= 0; (* write the closing byte for the string *)

(* revision history

ks	6. dec. 2009 rev 1.0
	original version

*)

END_FUNCTION

// ---- beckhoff_network/POUs/CO_NVERT/SHA1_STR.TcPOU
FUNCTION_BLOCK SHA1_STR
VAR_INPUT
	RUN: BOOL;
END_VAR
VAR_OUTPUT
	DONE: BOOL;
END_VAR
VAR_IN_OUT
	STR: STRING(STRING_LENGTH);
	SHA1 : ARRAY [0..19] OF BYTE;
END_VAR

VAR
	run_last: BOOL;
	SHA1_STREAM : SHA1_STREAM;
	buf : ARRAY [0..63] OF BYTE;
	mode : INT;
	size : UDINT;
	pos : UDINT;
END_VAR

(*
version 1.0	06. dec. 2009
programmer 	ks
tested BY	ks

SHA1_STR berechnet den MD5 Hash eines Strings
*)

CASE mode OF
0:	(* Wait für Start *)
	IF RUN AND NOT run_last THEN
		DONE := FALSE;
		mode := 1; (* Initialisierung *)
		size := LEN(STR);
	END_IF;

2:	(* Data copy and Calc *)
	IF size > 0 THEN
		_STRING_TO_BUFFER(STR:=MID(STR, UDINT_TO_INT(SIZE), UDINT_TO_INT(POS) + 1), POS:=0, PT:=ADR(buf), SIZE:=SIZEOF(buf));
	END_IF;

3:	DONE := TRUE;
	mode := 0; (* Stop *)

END_CASE;

IF mode > 0 THEN
	SHA1_STREAM(SIZE:=size, MODE:=mode, BUF:=buf, SHA1:=SHA1, POS=>pos);
END_IF;

run_last := RUN;

(* revision history

ks	6. dec. 2009 rev 1.0
	original version

*)

END_FUNCTION_BLOCK

// ---- beckhoff_network/POUs/CO_NVERT/SHA1_STREAM.TcPOU
FUNCTION_BLOCK SHA1_STREAM
VAR_IN_OUT
	MODE : INT;
	BUF : ARRAY [0..63] OF BYTE;
	SHA1 : ARRAY [0..19] OF BYTE;
	SIZE : UDINT;
END_VAR

VAR_OUTPUT
	POS : UDINT;
END_VAR

VAR
	hash : ARRAY [0..4] OF DWORD;
	end : UDINT;
	block : UDINT;
	pad_1 : BOOL;
	w : ARRAY [0..79] OF DWORD;
	n : INT;
	n1 : INT;
	a : DWORD;
	b : DWORD;
	c : DWORD;
	d : DWORD;
	e : DWORD;
	f : DWORD;
	k : DWORD;
	x : DWORD;
	z : INT;
END_VAR

(*
version 1.0	06. dec. 2009
programmer 	ks
tested BY	ks

SHA1_STREAM berechnet den SHA1 Hash eines Datenstromes
*)

CASE MODE OF

1:	(* Initialisierung der Hash-Werte *)
	hash[0] := DWORD#16#67452301;
	hash[1] := DWORD#16#EFCDAB89;
	hash[2] := DWORD#16#98BADCFE;
	hash[3] := DWORD#16#10325476;
	hash[4] := DWORD#16#C3D2E1F0;

	(* Buffer initialisieren *)
	FOR n := 16 TO 79 DO
   		w[n] := DWORD#0;
	END_FOR;

	block := SHR(SIZE,6) + BOOL_TO_UDINT((UDINT_TO_BYTE(SIZE) AND 16#3F) > 55);	(* benötigte Blocks errechnen *)

	pad_1 := FALSE;
	POS := 0;
	End := SIZE;
	SIZE := MIN(64,End);
	MODE := 2;

2:	FOR n := UDINT_TO_INT(SIZE) TO 63 DO (* Fuell-Bytes anhängen *)
		BUF[n] := 0;
	END_FOR;

	IF SIZE < 64 AND NOT pad_1 THEN
		BUF[SIZE] := 2#1000_0000;
		pad_1 := TRUE;
	END_IF;

	POS := POS + SIZE;
	SIZE := MIN(64,End - POS);

	n := 0;	(* Byte-Array in DWORD-Array umkopieren *)
	FOR n1 := 0 TO 15 DO
		w[n1] := DWORD_OF_BYTE(BUF[n],BUF[n+1],BUF[n+2],BUF[n+3]);
		n := n + 4;
	END_FOR;

	IF block = 0 THEN (* am Ende des letzten Blocks die Datenlänge eintragen *)
		w[15] := SHL(UDINT_TO_DWORD(End),3); (* Anzahl Datenbits eintragen *)
		MODE := 3;
	ELSE
		block := block - 1;
	END_IF;

	FOR n := 16 TO 79 DO (* erweitern der 16 32-bit-Worte auf 80 32-bit-Worte *)
		w[n] := ROL(w[n-3] XOR w[n-8] XOR w[n-14] XOR w[n-16],1);
	END_FOR;

	a := hash[0];
	b := hash[1];
	c := hash[2];
	d := hash[3];
	e := hash[4];

	FOR n := 0 TO 79 DO
		IF n <= 19 THEN
			f := (b AND c) OR (NOT(b) AND d);
			k := DWORD#16#5A827999;
		ELSIF n <= 39 THEN
			f := b XOR c XOR d;
			k := DWORD#16#6ED9EBA1;
		ELSIF n <= 59 THEN
			f := (b AND c) OR (b AND d) OR (c AND d);
			k := DWORD#16#8F1BBCDC;
		ELSE
			f := b XOR c XOR d;
			k := DWORD#16#CA62C1D6;
		END_IF;

		x := ROL(a,5) + f + e + k + w[n];
		e := d;
		d := c;
		c := ROL(b,30);
		b := a;
		a := x;
	END_FOR;

	(* aktuelle Hash-Werte zum letzten Wert addieren *)
	hash[0] := hash[0] + a;
	hash[1] := hash[1] + b;
	hash[2] := hash[2] + c;
	hash[3] := hash[3] + d;
	hash[4] := hash[4] + e;

END_CASE;

IF MODE = 3 THEN
	z := 0;
	FOR n := 0 TO 4 DO (* konvertiere DWORD auf BYTE-Array *)
		FOR n1 := 0 TO 3 DO
			hash[n] := ROL(hash[n],8);
			SHA1[z] := DWORD_TO_BYTE(hash[n]);
			z := z + 1;
		END_FOR;
	END_FOR;
END_IF;

(* revision history

ks	6. dec. 2009 rev 1.0
	original version

*)

END_FUNCTION_BLOCK

// ---- beckhoff_network/POUs/CO_NVERT/URL_ENCODE.TcPOU
FUNCTION URL_ENCODE : STRING(STRING_LENGTH)
VAR_INPUT
	IN : STRING(STRING_LENGTH);
END_VAR
VAR
	pt_in : POINTER TO ARRAY[1..255] OF BYTE;
	pt_out : POINTER TO ARRAY[1..256] OF BYTE;
	pos_in : INT;
	pos_out : INT;
	stop : INT;
	tb : BYTE;
END_VAR


(*
version 1.1		10. may. 2010
programmer 	hugo
tested by		hugo

URL_ENCODE checks a string if it contains only non reserved characters for an url.
the non reserved characters are : [A..Z], [a..z], [0..9], -_.~
if reserved characters are found then these characters are converted to %HH while HH is the Hexadezimal representation of the character in Alphabetic Letters.
for example the reserved character # will be converted to '%23'.

*)

pt_in  := ADR(in);
pt_out := ADR(URL_ENCODE);

(* scan the input string and convert unallowed characters *)
pos_in := 1;
stop := LEN(in);
FOR pos_out := 1 TO 250 DO
	IF pos_in > stop THEN
		EXIT;
	ELSIF IS_URLCHR(pt_in^[pos_in]) THEN
		pt_out^[pos_out] := pt_in^[pos_in];
		(* increment in by 1 *)
		pos_in := pos_in + 1;
	ELSE
		(* cannot fit 3 digits, exit *)
		IF pos_out > 248 THEN EXIT; END_IF;
		(* invalid character that needs to be converted *)
		pt_out^[pos_out] := 37;    (* start with % sign *)
		pos_out := pos_out + 1;
		(* need to add the two hex digits *)
		tb := SHR(pt_in^[pos_in],4);
		IF tb > 9 THEN
			pt_out^[pos_out] := tb + 55;
		ELSE
			pt_out^[pos_out] := tb + 48;
		END_IF;
		pos_out := pos_out + 1;
		tb := pt_in^[pos_in] AND 16#0F;
		IF tb > 9 THEN
			pt_out^[pos_out] := tb + 55;
		ELSE
			pt_out^[pos_out] := tb + 48;
		END_IF;
		(* increment in and out because out has to move 3 digits *)
		pos_in := pos_in + 1;
	END_IF;
END_FOR;

(* terminate the output string *)
pt_out^[pos_out] := 0;

(* revision history
hm	27. apr. 2008	rev 1.0
	original version

ks	10. mai. 2008	rev 1.1
	stringlength 250

*)

END_FUNCTION

// ---- beckhoff_network/POUs/DEMO/CSV_PARSER_FILE_DEMO.TcPOU
PROGRAM CSV_PARSER_FILE_DEMO
VAR CONSTANT
	 line_cnt : INT:=2;
	 col_cnt : INT:=4;
END_VAR
VAR
	CPF : CSV_PARSER_FILE;
	FS : FILE_SERVER;
	FSD : FILE_SERVER_DATA;
	PT : NETWORK_BUFFER;
	filename : STRING;
	value :	STRING(STRING_LENGTH);
	sep : BYTE;
	step : INT;
	result : BYTE;
	offset : UDINT;
	run : BYTE;
	done : BOOL;
	value_real : REAL;
	cnt : INT;
	line : INT;
	idx : INT;
	data : ARRAY [1..line_cnt, 1..col_cnt] OF REAL;

	(*LOG_MSG : LOG_MSG;
	_debug_enable : BOOL := TRUE;*)
END_VAR

(* Demo-Programm: CSV-Datei mittels Enumeration auswerten

die groesse des arrays kann mittels konstanten line_cnt und col_cnt angepasst werden

 ----- den nachfolgenden Textblock als datei "csv.txt" auf der sps ablegen ---
10.45,20,30,40.8
115,3450.2123,456,123.1
---------------------------------------------------------------------------------*)

CASE step OF

00:	IF NOT done THEN
		filename := 'csv.txt'; (* File_Daten einrichten *)
		OFFSET := 0; (* Start Offset vorgeben *)
		FSD.AUTO_CLOSE := T#0ms; (* kein Automatisches schliessen *)
		sep :=44; (* Trennzeichen , *)
		run := 1; (* Element suchen *)
		cnt := 0;
		step := 20;
	END_IF;

20:	IF run = 0 THEN (* kein Befehl mehr aktiv ? *)
		(* ---------------------- Debug-Message ----------------------------*)
		(*IF _debug_enable THEN
			LOG_CL.NEW_MSG := 'CPFD: /value >~2< /offset ~3 /Run ~4 /Result ~5';
			LOG_CL.PRINTF[2] := value;
			LOG_CL.PRINTF[3] := UDINT_TO_STRING(OFFSET);
			LOG_CL.PRINTF[4] := BYTE_TO_STRING(run);
			LOG_CL.PRINTF[5] := BYTE_TO_STRING(result);
			LOG_MSG();
		END_IF;*)
		(* -----------------------------------------------------------------*)

		run := 1; (*  nächstes Element suchen  *)

		IF result = 1 OR result = 2 THEN
			(* automatische konvertierung in real ausführen *)
			IF LEN(value) <= 20 THEN
				value_real := FLOAT_TO_REAL(FLT:=value);
			ELSE
				value_real := 0.0;
			END_IF;

			cnt := cnt + 1;
			IF cnt <= line_cnt * col_cnt THEN
				line := (cnt / col_cnt) + 1;
				idx := (cnt MOD col_cnt);
				data[line,idx] := value_real; (* Daten in Array eintragen *)
			END_IF;

		ELSIF result = 10 THEN (* nichts mehr gefunden *)
			run := 0; (* keine weitere INI Auswertung erwünscht *)
			FSD.MODE := 5; (* Datei schliessen *)
			step := 30;
		END_IF;
	END_IF;

30:	IF FSD.MODE = 0 THEN (* Befehl Datei schliessen beendet *)
		step := 0;
		done := TRUE;
	END_IF;

END_CASE;

CPF(SEP:=sep,FILENAME:=FILENAME,FSD:=FSD,RUN:=run,OFFSET:=OFFSET,VALUE:=value,PT:=PT,RESULT=>result); (* CSV PARAMETER FILE *)
FS(FSD:=FSD,PT:=PT); (* FILE_SERVER *)

END_PROGRAM

// ---- beckhoff_network/POUs/HARDWARE/FILE_SERVER.TcPOU
FUNCTION_BLOCK FILE_SERVER
VAR_IN_OUT
	FSD : FILE_SERVER_DATA;
	PT : NETWORK_BUFFER;
END_VAR
VAR
	buf_size : UDINT;
	handle : UINT; (* Filehandle *)
	read_max_length : UDINT;(* maximale Datenlänge *)
	file_position : UDINT;(* aktueller Schreib/Lesezeiger *)
	used_filename : STRING;(* aktueller Dateiname *)
	close_time : TIME;
	length_read : UDINT;
	write_length : UDINT;
	length_written : UDINT;
	open_handle : UINT;
	seek_position : UDINT;
	seek_mode : INT;
	seek_data : ARRAY[0..1] OF DINT;
	tell_position : UDINT;
	open_mode : DWORD;
	last_mode: BYTE;
	command : BYTE;
	error_code : BYTE;
	error : BOOL;
	file_change : BOOL;
	step : INT;
	t_diff : TIME;
	tx_last : TIME;
	tx : TIME;
	X : FW_AdsRdWrt;
	tmpDW : UDINT;
	para : BOOL;

	(*LOG_MSG : LOG_MSG;
	_debug_enable : BOOL := TRUE;
	step_last : INT;*)
END_VAR

(*
version 1.0		23. sep. 2010
programmer 		ks
tested by			ks

FILE_SERVER ermöglicht den Zugriff auf Datteien mittels Plattform-Neutraler Schnittstelle
*)

(*
- Befehle -
1 = File_Open_Exist + File_Read
2 = File_Open_Exist + File_Write
3 = File_Open_New  + File_Write
4 = File_Remove
5 = File_Close

- Action -
1 = file_open (open)
2 = file_close (close)
3 = file_read (read)
4 = file_write (write)
5 = file_seek (setpos)
6 = file_tell (getpos)
7 = file_remove (delete)

---- fehlermeldungen----

00	Kein Fehler
19	SYSTEMSERVICE_FOPEN		Unbekannte oder ungültige Parameter
28	SYSTEMSERVICE_FOPEN		Datei nicht gefunden. Ungültiger Dateiname oder Dateipfad
38	SYSTEMSERVICE_FOPEN		Keine weiteren freien File Handles.
51	SYSTEMSERVICE_FCLOSE	ungültiges oder unbekanntes file handle.
62	SYSTEMSERVICE_FCLOSE	Datei wurde mit falscher Methode geöffnet.
67	SYSTEMSERVICE_FREAD		ungültiges oder unbekanntes file handle.
74	SYSTEMSERVICE_FREAD		Kein Speicher für Lesebuffer.
78	SYSTEMSERVICE_FREAD		Datei wurde mit falscher Methode geöffnet.
83	SYSTEMSERVICE_FWRITE	ungültiges oder unbekanntes file handle
94	SYSTEMSERVICE_FWRITE	Datei wurde mit falscher Methode geöffnet.
99	SYSTEMSERVICE_FSEEK		ungültiges oder unbekanntes file handle.
110	SYSTEMSERVICE_FSEEK		Datei wurde mit falscher Methode geöffnet.
115	SYSTEMSERVICE_FTELL		ungültiges oder unbekanntes file handle.
126	SYSTEMSERVICE_FTELL		Datei wurde mit falscher Methode geöffnet
140	SYSTEMSERVICE_FDELETE	Datei nicht gefunden. Ungültiger Dateiname oder Dateipfad.
255	Applikation					Position liegt hinter dem Dateiende

*)

(* read system timer *)
tx := UDINT_TO_TIME(T_PLC_MS());
t_diff := tx - tx_last;
tx_last := tx;

CASE step OF
0:
	IF FSD.MODE = LIMIT(1,FSD.MODE,5) THEN

		(* ---------------------- Debug-Message ----------------------------*)
		(*IF _debug_enable THEN
			LOG_CL.NEW_MSG := 'FS: File_Start Mode=~1';
			LOG_CL.PRINTF[1] := BYTE_TO_STRING(FSD.MODE);
			LOG_MSG();
		END_IF;*)
		(* -----------------------------------------------------------------------------*)

		(* Initialisierung *)
		X.sNetId := '';
		X.tTimeout := T#5s;
		X.nPort := 10000; (* AMSPORT_R3_SYSSERV *)

		buf_size := SIZEOF(PT.BUFFER);
		close_time := T#1ms; (* wenn Schritt aktiv ist, dann Close-Timer rücksetzen *)

		IF FSD.MODE = 4 THEN (* File_Remove *)
			IF handle > 0 THEN
				File_change := TRUE;
				step := 32000; (* File_Close ausführen *)
			ELSE
				step := 90; (* File_Remove ausführen *)
			END_IF;

		ELSIF FSD.MODE = 5 THEN (* File_Close *)
			step := 32000; (* File_Close ausführen *)

		ELSIF handle = 0 THEN (* MODE 1,2,3 *)
			step := 100; (* File muss erst geöffnet werden *)

		ELSE (* File ist geöffnset *)
			IF used_filename = FSD.FILENAME AND FSD.MODE = last_mode THEN (* kein Moduswechsel ? *)
				step := 200; (* ohne open prozedure weitermachen *)
			ELSE
				step := 32000;
				File_change := TRUE;
			END_IF;
		END_IF;

	ELSIF handle > 0 THEN (* offene Datei gefunden - AutoClose Modus *)
		IF FSD.AUTO_CLOSE > T#0s THEN
			close_time := close_time + t_diff; (* Close_Time hochzählen *)
			IF close_time > FSD.AUTO_CLOSE THEN (* Zeit überschrittenen *)
				step := 32000; (* automatisch Datei schliessen *)
			END_IF;
		END_IF;
	END_IF;

(* ----------------------------------- *)
090: (* File_Remove *)
	command := 7; (* File Remove *)
	step := 95;

095: (* File_Remove beendet *)
	IF command = 0 THEN
		step := 30000; (* Beenden *)
	END_IF;
(* ----------------------------------- *)

100: (* File_Open *)
	IF FSD.MODE = 3 THEN (* Open_New + File Write *)
		open_mode := 16#0001_001A; (* PATH_GENERIC + WRITEPLUS + BINARY *)
	ELSE (* Mode 1 Open_Exist + File _Read / Mode 2 Open_Exist + File_Write *)
		open_mode := 16#0001_0019; (* PATH_GENERIC + READPLUS + BINARY *)
	END_IF;
	command := 1; (* FileOpen *)
	step := 105;

105: (* File Open beendet *)
	IF command = 0 THEN
		IF error THEN
			step := 30000; (* Beenden *)
		ELSE
			(* Filedaten eintragen *)
			close_time := T#1ms; (* Timer freigeben *)
			handle := open_handle;
			used_filename := FSD.FILENAME;
			file_position := UDINT#4294967295; (* maximal = unbekannt *)
			last_mode := FSD.MODE;
			step := 110;
		END_IF;
	END_IF;

110: (* File Seek *)
	command := 5; (* File-Seek *)
	seek_position := 0;
	seek_mode := 2; (* SEEK_END - Seek from the end of file *)
	step := 115;

115: (* File Seek beendet *)
	IF command = 0 THEN
		IF error THEN
			step := 30000; (* Beenden *)
		ELSE
			command := 6; (* File-Tell starten *)
			step := 120;
		END_IF;
	END_IF;

120: (* File Tell beendet *)
	IF command = 0 THEN
		IF error THEN
			step := 30000; (* Beenden *)
		ELSE
			FSD.FILE_SIZE := tell_position; (* aktuelle Dateigroesse *)
			FSD.FILE_OPEN := TRUE;
			step := 200;
		END_IF;
	END_IF;

200: (* File Seek *)
	IF FSD.OFFSET > FSD.FILE_SIZE THEN (* prüfe auf gültige offset-vorgabe *)
		error_code := 255;
		step := 30000; (* Beenden *)
	ELSIF FSD.OFFSET <> file_position THEN
		command := 5; (* File-Seek *)
		seek_position := FSD.OFFSET;
		seek_mode := 0; (* Seek from beginning of file *)
		step := 210;
	ELSE
		step := 300;
	END_IF;

210: (* File Seek *)
	IF command = 0 THEN
		file_position := seek_position;
		IF error THEN
			step := 30000; (* Beenden *)
		ELSE
			step := 300;
		END_IF;
	END_IF;

300: (* Read or Write ? *)
	IF FSD.MODE = 1 THEN
		step := 400; (* Read *)
	ELSE
		step := 500; (* Write *)
	END_IF;

400: (* File Read *)
	IF UINT_TO_UDINT(PT.SIZE) > buf_size THEN (* Leselänge auf Buffergroesse begrenzen *)
		read_max_length := buf_size;
	ELSE
		read_max_length := UINT_TO_UDINT(PT.SIZE);
	END_IF;

	IF read_max_length > buf_size THEN
		read_max_length := buf_size;  (* Leselänge auf Buffergroesse begrenzen *)
	END_IF;

	(* Leselänge an Dateilänge anpassen *)
	IF file_position + read_max_length > FSD.FILE_SIZE THEN
		read_max_length := FSD.FILE_SIZE - file_position;
	END_IF;

	IF read_max_length > 0 THEN
		command := 3; (* File_Read *)
		step := 410;
	ELSE
		PT.SIZE := UINT#0;
		step := 30000; (* Beenden *)
	END_IF;

410: (* File Read *)
	IF command = 0 THEN
		PT.SIZE := UDINT_TO_UINT(length_read);
		IF NOT Error THEN
			file_position := file_position + length_read; (* aktueller File_Position korrigieren *)
			FSD.OFFSET := file_position;
		END_IF;
		step := 30000; (* Beenden *)
	END_IF;

500: (* File Write *)
	IF UINT_TO_UDINT(PT.SIZE) > buf_size THEN (* Schreiblänge auf Buffergroesse begrenzen *)
		write_length := buf_size;
	ELSE
		write_length := UINT_TO_UDINT(PT.SIZE);
	END_IF;

	IF write_length > 0 THEN
		command := 4; (* File_Write *)
		step := 510;
	ELSE
		step := 30000; (* Beenden *)
	END_IF;

510:
	IF command = 0 THEN
		IF NOT Error THEN
			file_position := file_position + length_written; (* aktueller File_Position korrigieren *)
			FSD.OFFSET := file_position;
			IF file_position > FSD.FILE_SIZE THEN (* Datei ist groesser geworden *)
				FSD.FILE_SIZE := file_position;
			END_IF;
		END_IF;
		step := 30000; (* Beenden *)
	END_IF;

 (* --------------------------------------------- *)

30000: (* Befehl fertig *)
	FSD.MODE := 0;
	FSD.ERROR := error_code;
	step := 0;

	(* ---------------- Debug-Message -----------------------*)
	(*IF _debug_enable THEN
		LOG_CL.NEW_MSG := 'FS: File_Stop: File ~1, error ~7, code ~8';
		LOG_CL.PRINTF[1]  := used_filename;
		LOG_CL.PRINTF[7]  := INT_TO_STRING(BOOL_TO_INT(error));
		LOG_CL.PRINTF[8]  := BYTE_TO_STRING(error_code);
		LOG_MSG();
	END_IF;*)
	(* --------------------------------------------- *)

32000:
	close_time := T#0s; (* Timer stoppen *)
	IF handle > 0 THEN
		command := 2; (* File_Close ausführen *)
	END_IF;
	step := 32100;

32100:
	IF command = 0 THEN (* File Close beendet *)
		(* Filedaten ablöschen *)
		FSD.FILE_OPEN := FALSE;
		file_position := 0;
		FSD.FILE_SIZE := 0;
		FSD.OFFSET := 0;
		used_filename := '';
		handle := 0;

		(* File_Name wurde fliegend geändert ? *)
		IF file_change THEN
			file_change := FALSE;
			step := 0;
		ELSE
			step := 30000;
		END_IF;
	END_IF;

END_CASE;

(* 1 = file_open
   2 = file_close
   3 = file_read
   4 = file_write
   5 = file_seek
   6 = file_tell
   7 = file_remove
*) 

X(bExecute := FALSE); (* Zyklischer FW_AdsRdWrt Aufruf *)

(* ------------ File Open ------------- *)
IF command = 1 THEN
	IF NOT para THEN
		para := TRUE;
		X(	nIdxGrp := 120, (* SYSTEMSERVICE_FOPEN *)
			nidxOffs := open_mode,
			cbWriteLen := SIZEOF(FSD.FILENAME),
			pWriteBuff := ADR(FSD.FILENAME),
			cbReadLen := SIZEOF(tmpDW),
			pReadBuff := ADR(tmpDW),
			bExecute := TRUE
			);
	ELSIF X.bBusy = FALSE THEN
		para := FALSE;
		error := X.bError;
		error_code := SEL(error,0,UDINT_TO_BYTE(X.nErrId + 16#10));

		IF X.cbRead >= SIZEOF(tmpDW) THEN
			open_handle := UDINT_TO_UINT(tmpDW);
		ELSE
			open_handle := 0;
		END_IF;
		command := 0;

		(* ---------------- Debug-Message -----------------------*)
		(*IF _debug_enable THEN
			LOG_CL.NEW_MSG := 'FS: Open: File ~1, handle ~2 , mode ~3 , error ~7, code ~8';
			LOG_CL.PRINTF[1] := FSD.FILENAME;
			LOG_CL.PRINTF[2] := DWORD_TO_STRING(open_handle);
			LOG_CL.PRINTF[3] := DWORD_TO_STRING(open_mode);
			LOG_CL.PRINTF[7] := INT_TO_STRING(BOOL_TO_INT(error));
			LOG_CL.PRINTF[8] := BYTE_TO_STRING(error_code);
			LOG_MSG();
		END_IF;*)
		(* -----------------------------------------------------------------*)
	END_IF;
END_IF;

(* ----------- File Close ------------- *)
IF command = 2 THEN
	IF NOT para THEN
		para := TRUE;
		X(	nIdxGrp := 121, (* SYSTEMSERVICE_FCLOSE *)
			nidxOffs := handle,
			cbWriteLen := 0,
			pWriteBuff := 0,
			cbReadLen := 0,
			pReadBuff := 0,
			bExecute := TRUE
			);
	ELSIF X.bBusy = FALSE THEN
		para := FALSE;
		error := X.bError;
		error_code := SEL(error,0,UDINT_TO_BYTE(X.nErrId + 16#30));
		command := 0;
		(* ---------------- Debug-Message -----------------------*)
		(*IF _debug_enable THEN
			LOG_CL.NEW_MSG := 'FS: Close: File ~1, error ~7, code ~8';
			LOG_CL.PRINTF[1] := used_filename;
			LOG_CL.PRINTF[7] := INT_TO_STRING(BOOL_TO_INT(error));
			LOG_CL.PRINTF[8] := BYTE_TO_STRING(error_code);
			LOG_MSG();
		END_IF;*)
		(* -----------------------------------------------------------------*)
	END_IF;
END_IF;

(* ------------ File Read ------------- *)
IF command = 3 THEN
	IF NOT para THEN
		para := TRUE;
		X(	nIdxGrp := 122, (* SYSTEMSERVICE_FREAD *)
			nidxOffs := handle,
			cbWriteLen := 0,
			pWriteBuff := 0,
			cbReadLen := read_max_length,
			pReadBuff := ADR(PT.BUFFER),
			bExecute := TRUE
			);
	ELSIF X.bBusy = FALSE THEN
		length_read := X.cbRead;
		para := FALSE;
		error := X.bError;
		error_code := SEL(error,0,UDINT_TO_BYTE(X.nErrId + 16#40));
		command := 0;

		(* ---------------- Debug-Message -----------------------*)
		(*IF _debug_enable THEN
			LOG_CL.NEW_MSG := 'FS: Read: File ~1, soll ~2,ist ~3 ,error ~7, code ~8';
			LOG_CL.PRINTF[1] := used_filename;
			LOG_CL.PRINTF[2] := UDINT_TO_STRING(read_max_length);
			LOG_CL.PRINTF[3] := UDINT_TO_STRING(length_read);
			LOG_CL.PRINTF[7] := INT_TO_STRING(BOOL_TO_INT(error));
			LOG_CL.PRINTF[8] := BYTE_TO_STRING(error_code);
			LOG_MSG();
		END_IF;*)
		(* -----------------------------------------------------------------*)
	END_IF;
END_IF;

(* ------------ File Write ------------- *)
IF command = 4 THEN
	IF NOT para THEN
		para := TRUE;
		X(	nIdxGrp := 123, (* SYSTEMSERVICE_FWRITE *)
			nidxOffs := handle,
			cbWriteLen := write_length,
			pWriteBuff := ADR(PT.BUFFER),
			cbReadLen := SIZEOF(length_written),
			pReadBuff := ADR(length_written),
			bExecute := TRUE
			);
	ELSIF X.bBusy = FALSE THEN
		para := FALSE;
		error := X.bError;
		error_code := SEL(error,0,UDINT_TO_BYTE(X.nErrId + 16#50));
		command := 0;

		(* ---------------- Debug-Message -----------------------*)
		(*IF _debug_enable THEN
			LOG_CL.NEW_MSG := 'FS: Write: File ~1, soll ~2,ist ~3 ,error ~7, code ~8';
			LOG_CL.PRINTF[1] := used_filename;
			LOG_CL.PRINTF[2] := UDINT_TO_STRING(write_length);
			LOG_CL.PRINTF[3] := UDINT_TO_STRING(length_written);
			LOG_CL.PRINTF[7] := INT_TO_STRING(BOOL_TO_INT(error));
			LOG_CL.PRINTF[8] := BYTE_TO_STRING(error_code);
			LOG_MSG();
		END_IF;*)
		(* -----------------------------------------------------------------*)
	END_IF;
END_IF;

(* ------------ File Seek ------------- *)
IF command = 5 THEN
	IF NOT para THEN
		para := TRUE;
		seek_data[0] := UDINT_TO_DINT(seek_position);
		seek_data[1] := INT_TO_DINT(seek_mode);

		X(	nIdxGrp := 124, (* SYSTEMSERVICE_FSEEK *)
			nidxOffs := handle,
			cbWriteLen := SIZEOF(seek_data),
			pWriteBuff := ADR(seek_data),
			cbReadLen := 0,
			pReadBuff := 0,
			bExecute := TRUE
			);
	ELSIF X.bBusy = FALSE THEN
		para := FALSE;
		error := X.bError;
		error_code := SEL(error,0,UDINT_TO_BYTE(X.nErrId + 16#60));
		command := 0;

		(* ---------------- Debug-Message -----------------------*)
		(*IF _debug_enable THEN
			LOG_CL.NEW_MSG := 'FS: Seek: File ~1,pos ~3 ,error ~7, code ~8';
			LOG_CL.PRINTF[1] := used_filename;
			LOG_CL.PRINTF[3] := UDINT_TO_STRING(seek_position);
			LOG_CL.PRINTF[7] := INT_TO_STRING(BOOL_TO_INT(error));
			LOG_CL.PRINTF[8] := BYTE_TO_STRING(error_code);
			LOG_MSG();
		END_IF;*)
		(* -----------------------------------------------------------------*)
	END_IF;
END_IF;

(* ------------ File Tell ------------- *)
IF command = 6 THEN
	IF NOT para THEN
		para := TRUE;
		X(	nIdxGrp := 125, (* SYSTEMSERVICE_FTELL *)
			nidxOffs := handle,
			cbWriteLen := 0,
			pWriteBuff := 0,
			cbReadLen := SIZEOF(tell_position),
			pReadBuff := ADR(tell_position),
			bExecute := TRUE
			);
	ELSIF X.bBusy = FALSE THEN
		para := FALSE;
		error := X.bError;
		error_code := SEL(error,0,UDINT_TO_BYTE(X.nErrId + 16#70));
		command := 0;

		(* ---------------- Debug-Message -----------------------*)
		(*IF _debug_enable THEN
			LOG_CL.NEW_MSG := 'FS: Tell: File ~1, pos ~3 ,error ~7, code ~8';
			LOG_CL.PRINTF[1] := used_filename;
			LOG_CL.PRINTF[3] := UDINT_TO_STRING(tell_position);
			LOG_CL.PRINTF[7] := INT_TO_STRING(BOOL_TO_INT(error));
			LOG_CL.PRINTF[8] := BYTE_TO_STRING(error_code);
			LOG_MSG();
		END_IF;*)
		(* -----------------------------------------------------------------*)
	END_IF;
END_IF;

(* ------------ File Remove ------------- *)
IF command = 7 THEN
	IF NOT para THEN
		para := TRUE;
		X(	nIdxGrp := 131, (* SYSTEMSERVICE_FDELETE *)
			nidxOffs := 16#0001_0000, (* PATH_GENERIC *)
			cbWriteLen := SIZEOF(FSD.FILENAME),
			pWriteBuff := ADR(FSD.FILENAME),
			cbReadLen := 0,
			pReadBuff := 0,
			bExecute := TRUE
			);
	ELSIF X.bBusy = FALSE THEN
		para := FALSE;
		error := X.bError;
		error_code := SEL(error,0,UDINT_TO_BYTE(X.nErrId + 16#80));
		command := 0;

		(* ---------------- Debug-Message -----------------------*)
		(*IF _debug_enable THEN
			LOG_CL.NEW_MSG := 'FS: Remove: File ~1, error ~7, code ~8';
			LOG_CL.PRINTF[1] := FSD.FILENAME;
			LOG_CL.PRINTF[7] := INT_TO_STRING(BOOL_TO_INT(error));
			LOG_CL.PRINTF[8] := BYTE_TO_STRING(error_code);
			LOG_MSG();
		END_IF;*)
		(* -----------------------------------------------------------------*)
	END_IF;
END_IF;

(* ---------------- Debug-Message -----------------------*)
(*IF _debug_enable THEN
	IF step_last <> step THEN
		LOG_CL.NEW_MSG := 'FS: Step: ~1';
		LOG_CL.PRINTF[1] := INT_TO_STRING(step);
		LOG_MSG();
	END_IF;
	step_last := step;
END_IF;*)
(* -----------------------------------------------------------------*)

(* revision history
ks	23. sep. 2010	rev 1.0
	original version
*)

END_FUNCTION_BLOCK

// ---- oscat_basic/POUs/Engineering/signal processing/OFFSET.TcPOU
FUNCTION OFFSET : REAL
VAR_INPUT
	X : REAL;
	O1, O2, O3, O4 : BOOL;
	D : BOOL;
END_VAR
VAR_INPUT CONSTANT
	Offset_1 : REAL;
	Offset_2 : REAL;
	Offset_3 : REAL;
	Offset_4 : REAL;
	default : REAL;
END_VAR

(*
version 1.0	12 jan 2007
programmer 	oscat
tested by	oscat

The Function offset adds offsets to an analog signal depending on digital inputs.
all selected offsets are added at the same time.
with the input D a default value instead of the input X can be used.

*)

IF D THEN OFFSET := default; ELSE OFFSET := X; END_IF;
IF O1 THEN OFFSET := OFFSET + offset_1; END_IF;
IF O2 THEN OFFSET := OFFSET + offset_2; END_IF;
IF O3 THEN OFFSET := OFFSET + offset_3; END_IF;
IF O4 THEN OFFSET := OFFSET + offset_4; END_IF;



(* revision history
hm	12. jan 2007
	original version


*)

END_FUNCTION

// ---- beckhoff_network/POUs/DEMO/DLOG_FILE_XML_DEMO.TcPOU
PROGRAM DLOG_FILE_XML_DEMO
VAR
	RTC_2: RTC_2;
	x : DLOG_DATA;
	DLOG_STORE_FILE_XML: DLOG_STORE_FILE_XML;
	CLK_PRG: CLK_PRG;
	cur_dt: DT;
	enable: BOOL := TRUE;
	rtc_set : BOOL := TRUE;

	trig_t : UDINT := 0;
	trig_m : BOOL;

	x1: DLOG_DT;
	x2 : DLOG_REAL;
	x3 : DLOG_DINT;
	x4 : DLOG_BOOL;
	x5: DLOG_STRING;
	GEN_SIN_1: GEN_SIN;
	COUNT_DR: COUNT_DR;
	error_c: DWORD;
	error_t: BYTE;
END_VAR

rtc_2(_in1 := rtc_set, _in2 := DT#2010-10-22-06:00:00);
cur_dt := rtc_2._out1;
rtc_set := FALSE;
clk_prg(_in1 := t#5s);
trig_m := clk_prg._out1;
x1(COLUMN := 'Timestamp', X := x); // DLOG_DT
GEN_SIN_1(_in1 := T#10m, _in2 := 100.0, _in3 := 50.0, _in4 := 0.0); // GEN_SIN
x2(VALUE := GEN_SIN_1._out2, N := 2, COLUMN := 'Sinus', X := x); // DLOG_REAL
COUNT_DR(_in3 := x.CLOCK_TRIG);
x3(VALUE := COUNT_DR._out1, COLUMN := 'Count', X := x); // DLOG_DINT
x4(STATE := COUNT_DR.CNT.2, OFF := 'OFF', ON := 'ON', COLUMN := 'Count_Bit_2', X := x); // DLOG_BOOL
x5(STR := DWORD_TO_STRB(COUNT_DR.CNT), COLUMN := 'Count_Hex', X := x); // DLOG_STRING
DLOG_STORE_FILE_XML(
    ENABLE := enable,
    TRIG_M := trig_m,
    TRIG_T := trig_t,
    FILENAME := 'test_#R.xml',
    DTI := cur_dt,
    X := x);
error_c := DLOG_STORE_FILE_XML.ERROR_C;
error_t := DLOG_STORE_FILE_XML.ERROR_T;

END_PROGRAM

// ---- oscat_basic/POUs/Engineering/signal generators/GEN_SIN.TcPOU
FUNCTION_BLOCK GEN_SIN
VAR_INPUT
	PT : TIME;
	AM : REAL := 1.0;
	OS : REAL;
	DL : REAL;
END_VAR
VAR_OUTPUT
	Q : BOOL;
	Out : REAL;
END_VAR
VAR
	tx : TIME;
	last : TIME;
	init : BOOL;
	temp : REAL;
END_VAR

(*
version 1.6	11. mar. 2009
programmer 	oscat
tested BY	oscat

this signal generator generates a sine wave output. The sine wave signal is defined by period time (PT), 
amplitude (AM), offset (OS) and a specific delay for the output signal (DL).
The Output waveform will have its max peak at AM/2 + OS and its minimum peak at -AM/2 + OS. 
The delay input can delay a signal up to PT, this can be useful to synchronize different generators 
and generate interleaving signals. A Cos wave can be generated accordingly.
in addition to a analog output Out there is a second boolean output Q with the corresponding binary signal.
*)

(* read system time and prepare input data *)
tx := DWORD_TO_TIME(T_PLC_MS()) - last;
DL := MODR(dl,1.0);
IF dl < 0.0 THEN dl := 1.0 - dl; END_IF;

(* init section *)
IF NOT init THEN
	init := TRUE;
	last := tx;
	tx := t#0s;
END_IF;

(* add last if one cycle is finished *)
IF tx >= pt THEN
	last := last + pt;
	tx := tx - pt;
END_IF;

(* generate sine wave *)
IF pt > t#0s THEN temp := SIN(math.PI2 * DWORD_TO_REAL(TIME_TO_DWORD(tx + MULTIME(pt, dl))) / DWORD_TO_REAL(TIME_TO_DWORD(pt))); END_IF;
out := am * 0.5 *  temp + os;

(* boolean output Q *)
q := NOT SIGN_R(temp);

(* revision history
hm	22. jan 2007	rev 1.0
	original version

hm	17 sep 2007	rev 1.1
	replaced time() with t_plc_ms for compatibilitx reasons

hm	27. nov 2007	rev 1.2
	avoid divide by 0 when pt = 0

hm	6. jan 2008		rev 1.3
	improved performance

hm	16. mar. 2008	rev 1.4
	added type conversion to avoid warnings under codesys 3.0

hm	18. oct. 2008	rev 1.5
	using math constants

hm	11. mar. 2009	rev 1.6
	changed real constants to use dot syntax

*)

END_FUNCTION_BLOCK

// ---- oscat_basic/POUs/Mathematical/SIGN_R.TcPOU
FUNCTION SIGN_R : BOOL
VAR_INPUT
	in : REAL;
END_VAR


(*
version 1.4	10. mar. 2009
programmer 	hugo
tested by		tobias

this function return true if the real input is negative

*)

SIGN_R := in < 0.0;


(* revision history
hm 19.1.2007	rev 1.1
	changed method of function for better compatibility to other systems

hm	1.12.2007	rev 1.2
	changed code to improve performance

hm	14. jun. 2008	rev 1.3
	improved performace

hm 10. mar. 2009	rev 1.4
	real constants updated to new systax using dot																																																																																																																																																																																																																																																																																																																																																																																																																																																																																																																																																																																																																																																																																																																																																																																																																																																																																																																																																																																																																																																											

*)

END_FUNCTION

// ---- oscat_basic/POUs/Logic/FF edge triggered/COUNT_DR.TcPOU
FUNCTION_BLOCK COUNT_DR
VAR_INPUT
	SET : BOOL;
	IN : DWORD;
	UP : BOOL;
	DN : BOOL;
	STEP : DWORD := 1;
	MX : DWORD := 16#FFFFFFFF;
	RST : BOOL;
END_VAR
VAR_OUTPUT
	CNT : DWORD;
END_VAR
VAR
	last_up: BOOL;
	last_dn: BOOL;
END_VAR

(*
	version 1.1	20. jan. 2011
	programmer 	hugo
	tested BY		tobias

Count_DR is a DWORD counter with independen up and dn inputs. the counter counts from 0 to mx and continues at 0 after is has reached mx
a step input sets the counters stepping width.

*)

IF rst THEN
	cnt := 0;
ELSIF set THEN
	cnt := LIMIT(0,in,mx);
ELSIF up AND NOT last_up THEN
	IF STEP > MX - CNT THEN
		CNT := CNT - MX + STEP - 1;
	ELSE
		CNT := CNT + STEP;
	END_IF;
ELSIF dn AND NOT last_dn THEN
	IF STEP > CNT THEN
		CNT := CNT - STEP + MX + 1;
	ELSE
		CNT := CNT - STEP;
	END_IF;
END_IF;
last_up := up;
last_dn := dn;

(* revision history
hm	12. jun 2008	rev 1.0
	original version

hm	20. jan. 2011	rev 1.1
	corrected init value of MX to 16#FFFFFFFF

*)

END_FUNCTION_BLOCK

// ---- beckhoff_network/POUs/DEMO/DNS_DYN_DEMO.TcPOU
PROGRAM DNS_DYN_DEMO
VAR
	DNS_DYN : DNS_DYN;
	IP_C : IP_C;
	S_BUF : NETWORK_BUFFER;
	R_BUF : NETWORK_BUFFER;
	IP_CONTROL : IP_CONTROL;
	enable: BOOL;
	done : BOOL;
	error_c : DWORD;
	error_t : BYTE;
	busy : BOOL;
	COUNT_DR: COUNT_DR;
	z: DWORD;

	GET_WAN_IP : GET_WAN_IP;
	t1: TON;
	done2 : BOOL;
	error_c2 : DWORD;
	error_t2 : BYTE;
	update : BOOL;
	new_ip: BOOL;
	wan_ip4: DWORD;
END_VAR
VAR // added by the converter: edge detectors and wires of the graphical bodies
    _w1 : ANY;
END_VAR

DNS_DYN(
    ENABLE := enable,
    UPDATE := update,
    T_UPDATE := t#0ms,
    MODE := 2,
    HOSTNAME := 'test.dyndns.org',
    USERNAME := 'test',
    PASSWORD := 'test',
    IP4 := wan_ip4,
    IP_C := IP_C,
    S_BUF := S_BUF,
    R_BUF := R_BUF);
busy := DNS_DYN.BUSY;
done := DNS_DYN.DONE;
error_c := DNS_DYN.ERROR_C;
error_t := DNS_DYN.ERROR_T;
// IP-Adresse des DNS-Server oder des DSL-Router
_w1 := DWORD_OF_BYTE(8, 8, 8, 8);
IP_CONTROL(IP := _w1, TIME_OUT := T#1s, IP_C := IP_C, S_BUF := S_BUF, R_BUF := R_BUF);
COUNT_DR(_in3 := done);
z := COUNT_DR._out1;
wan_ip4 := GET_WAN_IP.WAN_IP4;
t1(IN := NOT t1.Q, PT := t#30s); // TON
GET_WAN_IP(ACTIVATE := t1.Q, IP_C := IP_C, S_BUF := S_BUF, R_BUF := R_BUF);
done2 := GET_WAN_IP.DONE;
new_ip := GET_WAN_IP.NEW_IP4;
error_c2 := GET_WAN_IP.ERROR_C;
error_t2 := GET_WAN_IP.ERROR_T;

END_PROGRAM

// ---- beckhoff_network/POUs/HARDWARE/IP_CONTROL.TcPOU
FUNCTION_BLOCK IP_CONTROL
VAR_IN_OUT
	IP_C : IP_C; (* IP_Control Verwaltungsstruktur *)
	S_BUF : NETWORK_BUFFER; (* Externer Sendbuffer *)
	R_BUF : NETWORK_BUFFER; (* Externer Receivebuffer *)
END_VAR
VAR_INPUT
	IP : DWORD; (* IP Adresse *)
	PORT : WORD; (* Port Nummer *)
	TIME_OUT : TIME; (* Ueberwachungszeit Connect / Send / Receive *)
END_VAR
VAR
	c_time : UDINT; (* CONNECT-Time (Zeit bei nicht vorhandener Verbindung) *)
	s_time : UDINT; (* SEND-Time    (Zeit seit letzten Datensenden) *)
	r_time : UDINT; (* RECEIVE-Time (Zeit seit letztem Datenempfang) *)

	c_enable : BOOL; (* Connect: freigabe *)
	c_ip : DWORD; (* Connect: aktuelle IP-Adresse *)
	c_ip_str : STRING(15);
	c_port : WORD; (* Connect: aktuelle Port-Nummer *)
	c_mode : BYTE; (* Connect: aktueller Mode UDP/TCP...... *)
	c_status : BYTE; (* Connect: Status (Errorcode) *)
	c_ready : BOOL; (* Connect: Verbindung aufgebaut *)
	c_ready_old : BOOL; (* Connect: letzter Zustand von c_ready für Flankenauswertung *)

	s_total : INT; (* Send: Gesamtanzahl Bytes zum senden *)
	s_cur_pos : INT; (* Send: aktuelle Sendeposition *)
	s_cur_size : INT; (* Send: aktuelle Sendegroesse *)
	s_max_size : INT; (* Send: maximale Telegrammlänge fuer Senden *)
	s_active : BOOL; (* Send: Daten senden ist aktiv *)
	s_status : BYTE; (* Send: Status (Errorcodes) *)
	s_ip_str : STRING(15);
	s_ip_exist : BOOL;

	r_status : BYTE; (* Receive: Status (Errorcodes) *)
	r_count : INT; (* Receive: Anzahl empfangener Bytes *)
	r_offset : INT; (* Receive: aktuelle Position in externen Receivebuffer *)
	r_max_size : INT; (* Receive: groesse des externen Empfangbuffers*)

	new_connection : BOOL; (* Neue Verbindungsparameter vorhanden *)
	tx : DWORD; (* letzter zeitwert *)
	error_time : DWORD; (* aktueller Timeout-Wert *)

	state: BYTE; (* schrittmerker für connect *)
	bytes_received : DINT;
	udp_mode : BOOL;

	socket : T_HSOCKET;
	server : T_HSOCKET;
	fbCreate	: FB_SocketUdpCreate;
	fbConnect : FB_SocketConnect;
	fbClose : FB_SocketClose;
	fbSendTo : FB_SocketUdpSendTo;
	fbReceiveFrom : FB_SocketUdpReceiveFrom;
	fbSend : FB_SocketSend;
	fbReceive : FB_SocketReceive;
	fbListen : FB_SocketListen;
	fbAccept : FB_SocketAccept;
	nErrId : UDINT;
	Send_Busy : BOOL;
	Send_Error : BOOL;
	Send_ErrId : UDINT;

	IPCR : IP_CONTROL_RESET;

	(*LOG_MSG : LOG_MSG;
	_debug_enable : BOOL := TRUE;
	debug_index : INT;
	debug_ID : INT;
	debug_lasterror : DWORD;
	state_last : INT;
	debug_last_id : INT := 255;*)

END_VAR

VAR CONSTANT
	STOP : BYTE := 0;
	UDP_INIT : BYTE:= 31;
	UDP_INIT_WAIT : BYTE:= 32;
	TC_INIT : BYTE := 51;
	TC_CONNECT : BYTE:= 52;
	TS_INIT : BYTE:= 53;
	TS_LISTEN_WAIT : BYTE:= 54;
	TS_ACCEPT : BYTE:= 55;
	TS_ACCEPT_WAIT : BYTE:= 56;
	C_CLOSE : BYTE := 190;
	C_CLOSE_WAIT : BYTE:= 191;
	C_CLOSE2 : BYTE := 192;
	C_CLOSE_WAIT2 : BYTE:= 193;
	C_WAIT : BYTE := 200;
	C_REC : BYTE := 210;
	C_REC_WAIT : BYTE := 211;
	C_SND : BYTE := 220;
	C_SND_WAIT1 : BYTE := 221;
	C_SND_WAIT2 : BYTE := 222;
END_VAR

(*

version 1.8		26. july. 2011
programmer 		ks
tested by			ks

IP_CONTROL ist ein Wrapper-Baustein um eine Hersteller neutrale Schnittstelle zum Ethernet zu schaffen



TYP 	TCP / UDP 	Aktiv / Passiv 		Port-Nummer erforderlich 	IP-Adresse erforderlich
0 		TCP 		Aktiv 			Ja 						Ja
1 		UDP 		Aktiv 			Ja 						Ja
2 		TCP 		Passiv 			Ja 						Ja (Adresse des aktiven Partners)
3 		UDP 		Passiv 			Ja 						Ja (Adresse des aktiven Partners)
4 		TCP 		Passiv 			Ja 						Nein (beliebiger aktiver Partner wird akzeptiert)
5 		UDP 		Passiv 			Ja 						Nein (beliebiger aktiver Partner wird akzeptiert)

*)

(* Bei PLC reset oder Programm Download werden alle alten Verbindungen geschlossen *)
IPCR();
IF NOT IPCR.READY THEN RETURN; END_IF;

(*####################  DEBUG-MESSAGE  ###################################*)
(*IF _debug_enable THEN
	IF IP_C.FIFO.ID > BYTE#0 THEN (* nur wenn Teilnehmer ID's vorhanden sind *)
		debug_index := IP_C.FIFO.NR;
		debug_ID := BYTE_TO_INT(IP_C.FIFO.X[debug_index]);
	END_IF;
END_IF;*)
(*########################################################################*)

(* read system time *)
tx := T_PLC_MS();

IF IP_C.C_PORT = 0 THEN
	IP_C.C_PORT := PORT; (* uebergebenen PORT durch parametrierten PORT ersetzen *)
END_IF;
IF IP_C.C_IP = 0 AND IP_C.C_MODE < 4 THEN
	IP_C.C_IP := IP; (* uebergebene IP durch paramtrierte IP ersetzen *)
END_IF;

new_connection := c_ip <> IP_C.C_IP OR c_mode <> IP_C.C_MODE OR c_port <> IP_C.C_PORT; (* neue Verbindungs erwünscht ? *)
c_enable := IP_C.C_ENABLE AND NOT new_connection;

IF IP_C.C_ENABLE AND IP_C.ERROR = 0 AND state = STOP THEN (* Freigabe,kein Fehler,kein Socket offen *)
	c_ip   := IP_C.C_IP;
	c_mode := IP_C.C_MODE;
	c_port := IP_C.C_PORT;
	c_ip_str := IP4_TO_STRING(c_ip);
	udp_mode := C_MODE.0; (* Mode 1,3,5 = udp *)

	error_time := TIME_TO_DWORD(MAX(T#200ms,TIME_OUT));
	IP_C.TIME_RESET := TRUE; (* Alle Timer ruecksetzen *)
	r_max_size := SIZEOF(R_BUF.BUFFER);
	s_max_size := SIZEOF(S_BUF.BUFFER);

	IF udp_mode THEN (* Mode: 1,3,5 = UDP CLIENT/SERVER *)
		state := UDP_INIT;
	ELSIF c_mode = 0 THEN (* Mode: 0 = TCP CLIENT *)
		state := TC_INIT;
	ELSE
		state := TS_INIT; (* Mode: 2,4 = TCP SERVER *)
	END_IF;

	IF c_mode < 5 THEN (* Empfänger-IP vorgeben *)
		s_ip_str := c_ip_str;
		s_ip_exist := TRUE;
	ELSE
		s_ip_str := '';
		s_ip_exist := FALSE;
	END_IF;

    	(*####################  DEBUG-MESSAGE  ###################################*)
	(*IF _debug_enable THEN
		LOG_CL.NEW_MSG := 'IP_CON: MODE ~1 / IP ~2 / PORT ~3 /ID ~6';
		LOG_CL.PRINTF[1] := BYTE_TO_STRING(C_MODE);
		LOG_CL.PRINTF[2] := IP4_TO_STRING(c_ip);
		LOG_CL.PRINTF[3] := WORD_TO_STRING(c_port);
		LOG_CL.PRINTF[6] := INT_TO_STRING(debug_ID);
		LOG_MSG();
	END_IF;*)
	(*########################################################################*)

END_IF;

(*####################  DEBUG-MESSAGE  ###################################*)
(*IF  _debug_enable THEN
	IF state <> state_last THEN
		LOG_CL.NEW_MSG := 'IP_STEP ~1 -IP_ID ~6';
		LOG_CL.PRINTF[1] := BYTE_TO_STRING(state);
		LOG_CL.PRINTF[6] := INT_TO_STRING(debug_ID);
		LOG_MSG();
		state_last := state;
	END_IF;
END_IF;*)
(*########################################################################*)

IF IP_C.TIME_RESET THEN (* Alle Timer ruecksetzen *)
	IP_C.TIME_RESET := FALSE; (* Reset rücksetzen *)
	c_time := tx; (* Connect Timer ruecksetzen *)
	s_time := tx; (* Send Timer ruecksetzen *)
	r_time := tx; (* Receive Timer ruecksetzen *)

	c_status := BYTE#0; (* letzten Connect Fehler rücksetzen *)
	s_status := BYTE#0; (* letzten Send Fehler rücksetzen *)
	r_status := BYTE#0; (* letzten Receive Fehler rücksetzen *)
END_IF;

(* ---------------------------------------------- *)

CASE state OF

UDP_INIT: (* UDP_CLIENT + SERVER *)
	(* 1. bei UDP-Client wird als lokalport 0 vorgegeben, damit das System automatisch einen freien lokalen Port sucht
	    2. bei UDP Server muss der gewüschte lokalport verwendet werden *)

	fbCreate(bExecute := FALSE);
	fbCreate(	bExecute := TRUE , sSrvNetId := '', sLocalHost := '', nLocalPort := SEL(c_mode = 1,c_port,0) , tTimeOut := TIME_OUT);
	fbCreate.bExecute := FALSE; (* vorbelegung *)
	state := UDP_INIT_WAIT;

UDP_INIT_WAIT:
	fbCreate();
	IF NOT fbCreate.bBusy THEN
		IF NOT fbCreate.bError THEN
			socket := fbCreate.hSocket;
			c_ready := TRUE; (* Connected *)
			state := C_WAIT;
		ELSE
			c_status := 1; (* FB_SocketUdpCreate failed *)
			nErrId := fbCreate.nErrId;
			state := C_CLOSE;
		END_IF;
	END_IF;

(* ---------------------------------------------- *)
TC_INIT: (* TCP-CLIENT (AKTIV) *)
	fbConnect(bExecute := FALSE);
	fbConnect(bExecute := TRUE, sSrvNetId := '', sRemoteHost := c_ip_str, nRemotePort := c_port, tTimeout := TIME_OUT);
	fbConnect.bExecute := FALSE; (* vorbelegung *)
	state := TC_CONNECT;

(* ---------------------------------------------- *)
TC_CONNECT:
	IF NOT c_enable OR c_status = 255 THEN (* keine freigabe oder connect timeout *)
		state := C_CLOSE;
	END_IF;

	fbConnect();
	IF NOT fbConnect.bBusy THEN
		IF fbConnect.bError THEN
			nErrID := fbConnect.nErrId;
			state :=TC_INIT; (* Nochmals versuchen *)
		ELSE
			socket := fbConnect.hSocket;
			c_ready := TRUE; (* Connected *)
			state := C_WAIT;
		END_IF;
	END_IF;
(* ---------------------------------------------- *)
TS_INIT: (* TCP-SERVER (PASSIV) *)
	fbListen(bExecute := FALSE);
	fbListen(bExecute := TRUE , sSrvNetId:= '' , sLocalHost:= '' , nLocalPort:= c_port , tTimeout:= TIME_OUT);
	fbListen.bExecute := FALSE;
	state := TS_LISTEN_WAIT;
(* ---------------------------------------------- *)
TS_LISTEN_WAIT:
	fbListen();
	IF NOT fbListen.bBusy THEN
		IF fbListen.bError THEN
			c_status := 3; (* FB_SocketListen failed *)
			nErrID := fbListen.nErrId;
			state := C_CLOSE;
		ELSE
			server := fbListen.hListener;
			state := TS_ACCEPT;
		END_IF;
	END_IF;
(* ---------------------------------------------- *)
TS_ACCEPT:
	fbAccept(bExecute := FALSE);
	fbAccept(bExecute := TRUE, sSrvNetId := '', hListener := server, tTimeout := TIME_OUT);
	fbAccept.bExecute := FALSE;
	state := TS_ACCEPT_WAIT;
(* ---------------------------------------------- *)
TS_ACCEPT_WAIT:
	fbAccept();
	IF NOT fbAccept.bBusy THEN

		state := TS_ACCEPT; (* vorbelegung  *)

		IF fbAccept.bError THEN
			c_status := 4; (* FB_SocketAccept failed *)
			nErrID := fbAccept.nErrId;
			state := C_CLOSE;
		ELSE (* no error *)
			IF fbAccept.bAccepted THEN
				socket := fbAccept.hSocket;
				IF socket.remoteAddr.sAddr  <> c_ip_str AND c_mode <> 4 THEN
					state := C_CLOSE; (* Remote ablehnen - Verbindung beenden *)
				ELSE
					state := C_WAIT;
					c_ready := TRUE; (* Connected *)
				END_IF;
			END_IF; (* fbAccept.bAccepted *)
		END_IF; (* NOT fbAccept.bError *)
	END_IF; (*  NOT fbAccept.bBusy *)
(* ---------------------------------------------- *)
C_CLOSE:
	c_ready := FALSE;
	IF socket.handle > 0 THEN
		fbClose(bExecute := FALSE );
		fbClose(bExecute := TRUE, sSrvNetId := '',	hSocket := socket);
		fbClose.bExecute := FALSE;
		state := C_CLOSE_WAIT;
	ELSE
		state:= C_CLOSE2;
	END_IF;

C_CLOSE_WAIT:
	fbClose();
	IF NOT fbClose.bBusy THEN
		socket := TCPADS_NULL_HSOCKET; (* Socket rücksetzen *)
		nErrId:= SEL(fbClose.bError,0,fbClose.nErrId);
		state:= C_CLOSE2;
	END_IF;

C_CLOSE2:
	IF server.handle > 0 THEN
		fbClose(bExecute := FALSE );
		fbClose(bExecute := TRUE, sSrvNetId := '',	hSocket := server);
		fbClose.bExecute := FALSE;
		state := C_CLOSE_WAIT2;
	ELSE
		state:= STOP;
	END_IF;

C_CLOSE_WAIT2:
	fbClose();
	IF NOT fbClose.bBusy THEN
		server := TCPADS_NULL_HSOCKET; (* Socket rücksetzen *)
		nErrId:= SEL(fbClose.bError,0,fbClose.nErrId);
		state:= STOP;
	END_IF;

(* ---------------------------------------------- *)

C_WAIT: (* Warten auf Anforderung für Beenden *)
	IF NOT c_enable OR NOT c_ready THEN
		state:= C_CLOSE;
	ELSIF S_BUF.SIZE > 0 AND IP_C.MAILBOX[2] = 0 AND s_ip_exist THEN
		state:= C_SND;
	ELSIF IP_C.MAILBOX[3] = 0 THEN
		state:= C_REC;
	END_IF;

(* ---------------------------------------------- *)

C_REC: (* Daten empfangen *)
	IF R_BUF.SIZE >= INT_TO_UINT(r_max_size) THEN
		R_BUF.SIZE := UINT#0;
		r_status := 254; (* Empfangsbuffer wegen Überlauf rückgesetzt *)
	END_IF;

	r_offset := SEL(udp_mode,UINT_TO_INT(R_BUF.SIZE),0);
	r_count := r_max_size - r_offset;
	bytes_received := 0;

	IF udp_mode THEN
		fbReceiveFrom(bExecute := FALSE );
		fbReceiveFrom(bExecute:= TRUE, sSrvNetId := '', hSocket:= socket, cbLen := r_count, pDest:= ADR(R_BUF.BUFFER), tTimeout:= TIME_OUT);
		fbReceiveFrom.bExecute := FALSE; (* Vorbelegung *)
	ELSE
		fbReceive(bExecute:= FALSE);
		fbReceive(bExecute:= TRUE, sSrvNetId := '' , hSocket:= socket , cbLen:= r_count, pDest:= ADR(R_BUF.BUFFER[r_offset]) , tTimeout:= TIME_OUT);
		fbReceive.bExecute:= FALSE;
	END_IF;
	state := C_REC_WAIT;

C_REC_WAIT:
	IF udp_mode THEN
		fbReceiveFrom(); (* UDP Mode *)
		IF NOT fbReceiveFrom.bBusy THEN
			IF NOT fbReceiveFrom.bError THEN
				IF fbReceiveFrom.nRecBytes > 0 THEN
					IF c_mode <> BYTE#5 AND fbReceiveFrom.sRemoteHost  <> c_ip_str THEN
						R_BUF.SIZE := UINT#0;
					ELSE
						bytes_received := fbReceiveFrom.nRecBytes;
						IF NOT s_ip_exist THEN
							s_ip_str := fbReceiveFrom.sRemoteHost;
							s_ip_exist := TRUE;
						END_IF;
					END_IF;
				END_IF;
				state := C_WAIT;
			ELSIF fbReceiveFrom.nErrId = 16#80072746 THEN (* Verbindung vom Remote beendet *)
				c_status := 253;
				c_ready := FALSE;
				state := C_WAIT;
			ELSE
				nErrId := fbReceiveFrom.nErrId;
				state := C_WAIT;
			END_IF;
		END_IF;
	ELSE
		fbReceive(); (* TCP Mode *)
		IF NOT fbReceive.bBusy THEN
			IF NOT fbReceive.bError THEN
				IF fbReceive.nRecBytes > 0 THEN
					bytes_received := fbReceive.nRecBytes;
				END_IF;
			ELSIF fbReceive.nErrId = 16#8004 THEN (* Verbindung vom Remote beendet *)
				c_status := 253;
				c_ready := FALSE;
			ELSE
				nErrId := fbReceive.nErrId;
			END_IF;
			state := C_WAIT;
		END_IF;
	END_IF;

	IF bytes_received > 0 THEN
		r_time := tx; (* Receive Timer ruecksetzen *)
		R_BUF.SIZE := INT_TO_UINT(r_offset + DINT_TO_UINT(bytes_received)); (* aktuelle buffersize eintragen *)
		IP_C.MAILBOX[1] := IP_C.MAILBOX[1] + 1; (* Receive Info *)
		IF IP_C.MAILBOX[1] = 0 THEN IP_C.MAILBOX[1] := 1; END_IF;
    		(*####################  DEBUG-MESSAGE  ###################################*)
		(*IF _debug_enable THEN
			LOG_CL.NEW_MSG := 'IP_REC DATA: POS: ~1 : SIZE: ~2 TOTAL ~3 -IP_ID ~6';
			LOG_CL.PRINTF[1] := INT_TO_STRING(r_offset);
			LOG_CL.PRINTF[2] := INT_TO_STRING(r_count);
			LOG_CL.PRINTF[3] := UINT_TO_STRING(R_BUF.SIZE);
			LOG_CL.PRINTF[6] := INT_TO_STRING(debug_ID);
			LOG_MSG();
		END_IF;*)
		(*########################################################################*)
	END_IF;

(* ---------------------------------------------- *)
C_SND:
	IF S_BUF.SIZE > 0 THEN
		IF c_ready AND c_enable THEN
			IF NOT s_active THEN
				s_total := LIMIT(0,UINT_TO_INT(S_BUF.SIZE),r_max_size); (* Gesamtanzahl an Bytes limitieren und uebergeben *)
				s_cur_pos  := 0;
				s_cur_size := 0;
				s_active := TRUE; (* Sende-Betrieb aktivieren *)
			END_IF;

			s_cur_pos := s_cur_pos + s_cur_size; (* neue Sende-Datenposition bestimmen *)
			IF s_total > s_cur_pos THEN (* weitere Daten zum senden vorhanden ? *)
				s_cur_size := s_total - s_cur_pos;
				s_cur_size := LIMIT(0, s_cur_size, s_max_size); (* Telegrammlänge begrenzen *)
				s_time := tx; (* Send Timer ruecksetzen *)
				r_time := tx; (* Receive Timer ruecksetzen *)
				state := C_SND_WAIT1;
			ELSE (* keine weitere Sendedaten vorhanden -> Senden beenden *)
				s_active := FALSE;
				S_BUF.SIZE := 0;
				state := C_WAIT;
			END_IF;
		END_IF;
	END_IF;

C_SND_WAIT1:
	IF udp_mode THEN
		fbSendTo(bExecute := FALSE );
		fbSendTo(bExecute := TRUE, sSrvNetId := '', hSocket := socket , cbLen := s_cur_size, pSrc := ADR(S_BUF.BUFFER[s_cur_pos]), sRemoteHost := s_ip_str, nRemotePort := c_port, tTimeout:= TIME_OUT);
		fbSendTo.bExecute := FALSE;
	ELSE
		fbSend(bExecute := FALSE);
		fbSend(bExecute := TRUE, sSrvNetId := '', hSocket := socket , cbLen:= s_cur_size, pSrc:=ADR(S_BUF.BUFFER[s_cur_pos]), tTimeout:= TIME_OUT);
		fbSend.bExecute := FALSE;
	END_IF;
	state := C_SND_WAIT2;

C_SND_WAIT2:
	IF udp_mode THEN
		fbSendTo();
		Send_Busy := fbSendTo.bBusy;
		Send_Error := fbSendTo.bError;
		Send_ErrId := fbSendTo.nErrId;
	ELSE
		fbSend();
		Send_Busy := fbSend.bBusy;
		Send_Error := fbSend.bError;
		Send_ErrId := fbSend.nErrId;
	END_IF;

	IF NOT Send_Busy THEN
		IF NOT Send_Error THEN
    			(*####################  DEBUG-MESSAGE  ###################################*)
			(*IF _debug_enable THEN
				LOG_CL.NEW_MSG := 'IP_SEN SEND_COUNT ~1 -IP_ID ~6';
				LOG_CL.PRINTF[1] := DINT_TO_STRING(s_cur_size);
				LOG_CL.PRINTF[6] := INT_TO_STRING(debug_ID);
				LOG_MSG();
			END_IF;*)
			(*########################################################################*)
			state := C_SND;
		ELSE
			nErrId := Send_ErrId;
			state := C_WAIT;
    			(*####################  DEBUG-MESSAGE  ###################################*)
			(*IF _debug_enable THEN
				LOG_CL.NEW_MSG := 'IP_SEN SEND ERROR ~1 -IP_ID ~6';
				LOG_CL.PRINTF[1] := UDINT_TO_STRING(nErrId);
				LOG_CL.PRINTF[6] := INT_TO_STRING(debug_ID);
				LOG_MSG();
			END_IF;*)
			(*########################################################################*)
		END_IF;
	END_IF;

END_CASE;

(* ---------------------------------------------- *)

IF c_ready THEN
	IF NOT c_ready_old THEN (* Verbindung aufgebaut - positive Flanke erkannt *)
		IP_C.C_STATE := 254;
		IP_C.TIME_RESET := TRUE; (* Alle Timer ruecksetzen *)
    		(*####################  DEBUG-MESSAGE  ###################################*)
		(*IF _debug_enable THEN
			LOG_CL.NEW_MSG := 'IP_CON: CONNECTED -IP_ID ~6';
			LOG_CL.PRINTF[6] := INT_TO_STRING(debug_ID);
			LOG_MSG();
		END_IF;*)
		(*########################################################################*)
	ELSE
		IP_C.C_STATE := 255; (* Verbindung ist aufgebaut *)
	END_IF;
ELSE
	IF c_ready_old THEN (* Verbindung abgebaut - negative Flanke erkannt *)
		IP_C.C_STATE := 1;
		IP_C.MAILBOX[1] := 0; (* Receive Info rücksetzen *)
		IP_C.MAILBOX[2] := 0; (* Send-Pause rücksetzen *)
		IP_C.MAILBOX[3] := 0; (* Receive-Pause rücksetzen *)
		IF NOT new_connection THEN
			s_active := FALSE; (* Sendeaktivitäten stoppen *)
			S_BUF.SIZE := 0; (* Sendelänge löschen *)
			(*IP_C.TIME_RESET := TRUE; *) (* Alle Timer ruecksetzen *)
		END_IF;
    		(*####################  DEBUG-MESSAGE  ###################################*)
		(*IF _debug_enable THEN
			LOG_CL.NEW_MSG := 'IP_CON: DISCONNECTED';
			LOG_MSG();
		END_IF;*)
		(*########################################################################*)

	ELSE
		IP_C.C_STATE := 0; (* Verbindung ist abgebaut *)
	END_IF;
END_IF;

c_ready_old := c_ready;

(* ---------------------------------------------- *)

IF IP_C.R_OBSERVE = FALSE OR s_active THEN
    r_time := tx;
END_IF;

IF c_status = 0 AND tx - c_time > error_time AND c_enable AND NOT c_ready AND c_mode < 2 THEN (* Connect Timeout *)
	c_status := 255; (* Timeout-Fehler ausgeben *)
END_IF;
IF s_status = 0 AND tx - s_time > error_time AND s_active THEN (* Send Timeout *)
	s_status := 255; (* Timeout-Fehler ausgeben *)
END_IF;
IF r_status = 0 AND tx - r_time > error_time AND c_ready AND IP_C.R_OBSERVE THEN (* Receive Timeout *)
	r_status := 255; (* Timeout-Fehler ausgeben *)
END_IF;

IP_C.ERROR := DWORD_OF_BYTE(c_status,s_status,r_status,0);

(*####################  DEBUG-MESSAGE  ###################################*)
(*IF  _debug_enable THEN
	IF (IP_C.ERROR <> debug_lasterror) THEN
		LOG_CL.NEW_MSG := 'IP_ERROR ~1 -IP_ID ~6';
		LOG_CL.PRINTF[1] := DWORD_TO_STRING(IP_C.ERROR);
		LOG_CL.PRINTF[6] := INT_TO_STRING(debug_ID);
		LOG_MSG();

		debug_lasterror := IP_C.ERROR;
		debug_last_id := debug_ID;
	END_IF;
END_IF;*)
(*########################################################################*)

(* revision history
ks	18. oct. 2008	rev 1.0
	original version
ks	05. jan. 2009	rev 1.1
	zusätzlichen Parameter "Port" hinzugefügt, und Code bei Verbindungsaufbau angepasst
ks	28. feb. 2009	rev 1.2
	connect code angepasst und verkürzung der zyklen bei Send
ks	20. oct. 2009	rev 1.3
	network_buffer basis 0
ks	06. dec. 2009	rev 1.4
	receive_count MAILBOX[1]
ks	10. nov. 2010	rev 1.5
	send_pause MAILBOX[2] and receive_pause MAILBOX[3] 
ks	07. feb. 2011	rev 1.6
	Fehlercode 253 bei Remote-Verbindungsabbruch 
ks	30. may. 2011	rev 1.7
	Fehler bei Empfangsüberwachung
ks	26. july. 2011	rev 1.8
	Error-Reset, diverse optimierungen 

*)

END_FUNCTION_BLOCK

// ---- beckhoff_network/POUs/HARDWARE/IP_CONTROL_RESET.TcPOU
FUNCTION_BLOCK IP_CONTROL_RESET
VAR_INPUT
END_VAR
VAR_OUTPUT
	READY : BOOL;
END_VAR
VAR
	fbSocketCloseAll : FB_SocketCloseAll;
	step : BYTE;
END_VAR

(* On PLC reset or program download close all old connections *)

CASE TCP_SERVER_RESET OF

2:	READY := TRUE;
	RETURN;

1:	IF step = 0 THEN
		RETURN;
	END_IF;

0:	TCP_SERVER_RESET := 1; (* Reset ist aktiv *)
	step := 1;

END_CASE;

CASE step OF

0:	RETURN;

1:	fbSocketCloseAll(sSrvNetId:= '', bExecute:= TRUE, tTimeout:= T#10s );
	step := 2;

2:	fbSocketCloseAll(bExecute:= FALSE);
	IF fbSocketCloseAll.bBusy = FALSE THEN
		step := 0;
		TCP_SERVER_RESET := 2; (* Reset durchgeführt , Bereit zur Verwendung *)
	END_IF;

END_CASE;

END_FUNCTION_BLOCK

// ---- beckhoff_network/POUs/NETWORK/GET_WAN_IP.TcPOU
FUNCTION_BLOCK GET_WAN_IP
VAR_IN_OUT
	IP_C : IP_C; (* IP_Control Verwaltungsstruktur *)
	S_BUF : NETWORK_BUFFER;
	R_BUF : NETWORK_BUFFER;
END_VAR
VAR_INPUT
	ACTIVATE : BOOL;
END_VAR
VAR_OUTPUT
	WAN_IP4 : DWORD;
	DONE : BOOL;
	NEW_IP4 : BOOL;
	ERROR_C : DWORD;
	ERROR_T : BYTE;
END_VAR
VAR
	URL_DATA : url;
	DNS_CLIENT : DNS_CLIENT;
	HTTP_GET : HTTP_GET;
	activate_last : BOOL;
	wan_ip4_last : DWORD;
	state : INT;
	st_ip : STRING(120);
	i1 :	INT;
	p1 : INT;
	p2 : INT;
	p3 : INT;
END_VAR

(*
version 1.1	28. dec. 2009
programmer 	ks
tested by	ks

GET_WAN_IP ermittelt die aktuelle WAN-IP (Internet-Adresse)
*)

CASE state OF

00:
	IF ACTIVATE AND NOT activate_last THEN
		state := 20;
		DONE := FALSE;
		ERROR_C := DWORD#0;
		ERROR_T := BYTE#0;
	END_IF;

20: (* URL for DNS UND HTTP-GET *)
	URL_DATA := STRING_TO_URL(STR:='checkip.dyndns.com',DEFAULT_PROTOCOL:='',DEFAULT_PATH:='');
	state := 40;

40:
	IF DNS_CLIENT.DONE THEN
		state := 60;
	ELSIF (DNS_CLIENT.ERROR > DWORD#00) THEN
		(* Fehlerbehandlung *)
		ERROR_C := DNS_CLIENT.ERROR;
		ERROR_T := BYTE#01;
		state := 100;
	END_IF;

60:
	IF HTTP_GET.DONE THEN
		state := 80;
	ELSIF (HTTP_GET.ERROR > DWORD#00) THEN
		(* Fehlerbehandlung *)
		ERROR_C := HTTP_GET.ERROR;
		ERROR_T := BYTE#02;
		state := 100;
	END_IF;

80:
	(* Als Antwort wird folgende HTML Seite empfangen , hier muss die IP-Adresse herauskopiert werden *)
	(* <html><head><title>Current IP Check</title></head><body>Current IP Address: 85.127.217.33</body></html> *)
	st_ip := '';
	p1 := 0;
	FOR i1 := UINT_TO_INT(HTTP_GET.BODY_START) TO UINT_TO_INT(HTTP_GET.BODY_STOP) DO
		IF R_BUF.BUFFER[i1] = BYTE#58 THEN (* suche ':' *)
			p1 := i1 + 2;
			EXIT;
		END_IF;
	END_FOR;

	p3 := p1 + 15;
	IF p1 > 0 AND p3 < UINT_TO_INT(HTTP_GET.BODY_STOP) THEN
		FOR p2 := p1 TO p3 DO
			IF R_BUF.BUFFER[p2] <> BYTE#60 THEN (* suche '<' *)
				st_ip := CONCAT(st_ip,CHR_TO_STRING(C:=R_BUF.BUFFER[p2]));
			ELSE
				EXIT;
			END_IF;
		END_FOR;
	END_IF;

	WAN_IP4 := IP4_DECODE(STR:=st_ip);

	IF WAN_IP4 <> DWORD#0 THEN
		DONE := TRUE;
		NEW_IP4 := WAN_IP4 <> wan_ip4_last;
		wan_ip4_last := WAN_IP4;
	ELSE
		ERROR_C := DWORD#01; (* keine gültige IP gefunden *)
		ERROR_T := BYTE#03;
	END_IF;
	state := 100;

100:
	(* UNLOCK HTTP DATA *)
	IF (NOT HTTP_GET.DONE) THEN
		state := 0;
		DONE := ERROR_T = BYTE#0;
	END_IF;

END_CASE;

(* ---------------- DNS --------------- *)
DNS_CLIENT(	IP_C:=IP_C,
			S_BUF:=S_BUF,
			R_BUF:=R_BUF,
			DOMAIN:=URL_DATA.DOMAIN,
			IP4_DNS:=DWORD#00,
			ACTIVATE:=state=40 (* DNS Start *)
			);
(* nicht oder nicht direkt verwendete Parameter *)
(* DWORD :=DNS_CLIENT.IP4;
   BOOL  :=DNS_CLIENT.DONE;
   BYTE  :=DNS_CLIENT.ERROR; *)
(* -------------------------------------*)

(* ------------- HTTP_GET --------------- *)

HTTP_GET(	IP_C:=IP_C,
			S_BUF:=S_BUF,
			R_BUF:=R_BUF,
			IP4:=DNS_CLIENT.IP4,
			GET:=state=60,
			MODE:=BYTE#2, (* HTTP 1.1 mit persistenter Verbindung *)
			UNLOCK_BUF:=state=100,
			URL_DATA:=URL_DATA
			);

(* nicht oder nicht direkt verwendete Parameter *)
(*STRING := HTTP_GET.HTTP_STATUS;
  UINT :=HTTP_GET.HEADER_START;
  UINT :=HTTP_GET.HEADER_STOP;
  UINT :=HTTP_GET.BODY_START;
  UINT :=HTTP_GET.BODY_STOP;
  BOOL :=HTTP_GET.DONE;
  BYTE :=HTTP_GET.ERROR;
*)
(* -------------------------------------*)

activate_last := ACTIVATE;

(* revision history
ks	28. dec 2009	rev 1.1
	original version

*)

END_FUNCTION_BLOCK

// ---- beckhoff_network/POUs/NETWORK/DNS_CLIENT.TcPOU
FUNCTION_BLOCK DNS_CLIENT
VAR_IN_OUT
	IP_C : IP_C; (* IP_Control Verwaltungsstruktur *)
	S_BUF : NETWORK_BUFFER;
	R_BUF : NETWORK_BUFFER;
END_VAR
VAR_INPUT
	ACTIVATE : BOOL;
	DOMAIN : STRING;
	IP4_DNS : DWORD;
END_VAR
VAR_OUTPUT
	IP4 : DWORD;
	DONE : BOOL;
	ERROR : DWORD;
END_VAR
VAR
	IP_FIFO : IP_FIFO;
	ip_state : BYTE;
	ip_id : BYTE;
	i : INT;
	state : INT;
	domain_copy : STRING;
	activate_last : BOOL;
	url_length : INT;
	char : BYTE;
	char_count : INT;
	tid : BYTE;
	anc : INT;
	x : BYTE;
	rr_stop : BOOL;
	ttl_last : DWORD;
	ttl_tmp : DWORD;

	(*LOG_MSG : LOG_MSG;
	_debug_enable : BOOL := TRUE;*)

END_VAR

(*
version 1.3	26. jul. 2011
programmer 	ks
tested BY	ks

DNS_CLIENT führt eine Domain-Name Abfrage bei einen DNS-Server durch

*)

(* Domain Name System (query) *)

CASE state OF

00:	IF ACTIVATE AND NOT activate_last THEN (* auf positive Flanke GET warten *)
		DONE := FALSE;
		ERROR := DWORD#0;
		state := 5;
	END_IF;

05:	IP4 := IP4_DECODE(str:=DOMAIN); (* prüfe ob domain schon eine IP4-Adresse ist *)
	IF IP4 > DWORD#00 THEN
		DONE := TRUE;
		state := 0;
        		(*####################  DEBUG-MESSAGE  ###################################*)
        		(*IF _debug_enable THEN
            		LOG_CL.NEW_MSG := 'DNS: S05 IP4 ~1';
            		LOG_CL.PRINTF[1]  := DOMAIN;
            		LOG_MSG();
        		END_IF;*)
        		(*########################################################################*)
	ELSE
		ip_state := BYTE#1;
		ttl_last := DWORD#0;
		domain_copy := DOMAIN; (* DOMAIN String sichern *)
		state := 10;
        		(*####################  DEBUG-MESSAGE  ###################################*)
        		(*IF _debug_enable THEN
            		LOG_CL.NEW_MSG := 'DNS: S05 START';
            		LOG_MSG();
        		END_IF;*)
        		(*########################################################################*)
	END_IF;

